 FB 134
BEGIN
   S703_TL_DC_PIN.Enable_Aux := FALSE;
   S703_TL_DC_PIN.Adv_Amount := 0;
   S703_TL_DC_PIN.Ret_Amount := 0;
   S703_TL_DC_PIN.LS_Adv1 := FALSE;
   S703_TL_DC_PIN.LS_Ret1 := FALSE;
   S703_TL_DC_PIN.LS_Adv2 := FALSE;
   S703_TL_DC_PIN.LS_Ret2 := FALSE;
   S703_TL_DC_PIN.LS_Adv3 := FALSE;
   S703_TL_DC_PIN.LS_Ret3 := FALSE;
   S703_TL_DC_PIN.LS_Adv4 := FALSE;
   S703_TL_DC_PIN.LS_Ret4 := FALSE;
   S703_TL_DC_PIN.LS_Adv5 := FALSE;
   S703_TL_DC_PIN.LS_Ret5 := FALSE;
   S703_TL_DC_PIN.LS_Adv6 := FALSE;
   S703_TL_DC_PIN.LS_Ret6 := FALSE;
   S703_TL_DC_PIN.LS_Adv7 := FALSE;
   S703_TL_DC_PIN.LS_Ret7 := FALSE;
   S703_TL_DC_PIN.LS_Adv8 := FALSE;
   S703_TL_DC_PIN.LS_Ret8 := FALSE;
   S703_TL_DC_PIN.SOL_Adv := FALSE;
   S703_TL_DC_PIN.SOL_Ret := FALSE;
   S703_TL_DC_PIN.M_Ready := FALSE;
   S703_TL_DC_PIN.T_CHK1 := T#0MS;
   S703_TL_DC_PIN.T_CHK2 := T#0MS;
   S703_TL_DC_PIN.PB_Lamp_CHK := FALSE;
   S703_TL_DC_PIN.PB_Error_Rst := FALSE;
   S703_TL_DC_PIN.M_FLICK := FALSE;
   S703_TL_DC_PIN.M_Adv_Err := FALSE;
   S703_TL_DC_PIN.M_Ret_Err := FALSE;
   S703_TL_DC_PIN.LP_Adv := FALSE;
   S703_TL_DC_PIN.LP_Ret := FALSE;
   S703_TL_DC_PIN.Visu_Adv := W#16#0;
   S703_TL_DC_PIN.Visu_Ret := W#16#0;
   S703_TL_DC_PIN.Error_T1.IN := FALSE;
   S703_TL_DC_PIN.Error_T1.PT := T#0MS;
   S703_TL_DC_PIN.Error_T1.Q := FALSE;
   S703_TL_DC_PIN.Error_T1.ET := T#0MS;
   S703_TL_DC_PIN.Error_T1.STATE := B#16#0;
   S703_TL_DC_PIN.Error_T1.STIME := T#0MS;
   S703_TL_DC_PIN.Error_T1.ATIME := T#0MS;
   S703_TL_DC_PIN.Error_T2.IN := FALSE;
   S703_TL_DC_PIN.Error_T2.PT := T#0MS;
   S703_TL_DC_PIN.Error_T2.Q := FALSE;
   S703_TL_DC_PIN.Error_T2.ET := T#0MS;
   S703_TL_DC_PIN.Error_T2.STATE := B#16#0;
   S703_TL_DC_PIN.Error_T2.STIME := T#0MS;
   S703_TL_DC_PIN.Error_T2.ATIME := T#0MS;
   S703_TL_DC_PIN.Adv_End_Aux := FALSE;
   S703_TL_DC_PIN.Ret_End_Aux := FALSE;
   S703_TL_DC_PIN.CHK_Aux1 := FALSE;
   S703_TL_DC_PIN.CHK_Aux2 := FALSE;
   S703_TL_DC_PIN.Error_T1_DN := FALSE;
   S703_TL_DC_PIN.Error_T2_DN := FALSE;
   S703_TL_DC_PIN.Adv_Memo := FALSE;
   S703_TL_DC_PIN.Visu_Adv_Arr[0] := FALSE;
   S703_TL_DC_PIN.Visu_Adv_Arr[1] := FALSE;
   S703_TL_DC_PIN.Visu_Adv_Arr[2] := FALSE;
   S703_TL_DC_PIN.Visu_Adv_Arr[3] := FALSE;
   S703_TL_DC_PIN.Visu_Adv_Arr[4] := FALSE;
   S703_TL_DC_PIN.Visu_Adv_Arr[5] := FALSE;
   S703_TL_DC_PIN.Visu_Adv_Arr[6] := FALSE;
   S703_TL_DC_PIN.Visu_Adv_Arr[7] := FALSE;
   S703_TL_DC_PIN.Visu_Adv_Arr[8] := FALSE;
   S703_TL_DC_PIN.Visu_Adv_Arr[9] := FALSE;
   S703_TL_DC_PIN.Visu_Adv_Arr[10] := FALSE;
   S703_TL_DC_PIN.Visu_Adv_Arr[11] := FALSE;
   S703_TL_DC_PIN.Visu_Adv_Arr[12] := FALSE;
   S703_TL_DC_PIN.Visu_Adv_Arr[13] := FALSE;
   S703_TL_DC_PIN.Visu_Adv_Arr[14] := FALSE;
   S703_TL_DC_PIN.Visu_Adv_Arr[15] := FALSE;
   S703_TL_DC_PIN.Visu_Ret_Arr[0] := FALSE;
   S703_TL_DC_PIN.Visu_Ret_Arr[1] := FALSE;
   S703_TL_DC_PIN.Visu_Ret_Arr[2] := FALSE;
   S703_TL_DC_PIN.Visu_Ret_Arr[3] := FALSE;
   S703_TL_DC_PIN.Visu_Ret_Arr[4] := FALSE;
   S703_TL_DC_PIN.Visu_Ret_Arr[5] := FALSE;
   S703_TL_DC_PIN.Visu_Ret_Arr[6] := FALSE;
   S703_TL_DC_PIN.Visu_Ret_Arr[7] := FALSE;
   S703_TL_DC_PIN.Visu_Ret_Arr[8] := FALSE;
   S703_TL_DC_PIN.Visu_Ret_Arr[9] := FALSE;
   S703_TL_DC_PIN.Visu_Ret_Arr[10] := FALSE;
   S703_TL_DC_PIN.Visu_Ret_Arr[11] := FALSE;
   S703_TL_DC_PIN.Visu_Ret_Arr[12] := FALSE;
   S703_TL_DC_PIN.Visu_Ret_Arr[13] := FALSE;
   S703_TL_DC_PIN.Visu_Ret_Arr[14] := FALSE;
   S703_TL_DC_PIN.Visu_Ret_Arr[15] := FALSE;
   S703_TL_DC_PIN.BLK_Move_Ret := 0;
   S703_TL_DC_PIN.Enable := FALSE;
   S703_TL_DC_PIN.Adv_End := FALSE;
   S703_TL_DC_PIN.Ret_End := FALSE;
   S703_TL_DC_LATCH1.Enable_Aux := FALSE;
   S703_TL_DC_LATCH1.Adv_Amount := 0;
   S703_TL_DC_LATCH1.Ret_Amount := 0;
   S703_TL_DC_LATCH1.LS_Adv1 := FALSE;
   S703_TL_DC_LATCH1.LS_Ret1 := FALSE;
   S703_TL_DC_LATCH1.LS_Adv2 := FALSE;
   S703_TL_DC_LATCH1.LS_Ret2 := FALSE;
   S703_TL_DC_LATCH1.LS_Adv3 := FALSE;
   S703_TL_DC_LATCH1.LS_Ret3 := FALSE;
   S703_TL_DC_LATCH1.LS_Adv4 := FALSE;
   S703_TL_DC_LATCH1.LS_Ret4 := FALSE;
   S703_TL_DC_LATCH1.LS_Adv5 := FALSE;
   S703_TL_DC_LATCH1.LS_Ret5 := FALSE;
   S703_TL_DC_LATCH1.LS_Adv6 := FALSE;
   S703_TL_DC_LATCH1.LS_Ret6 := FALSE;
   S703_TL_DC_LATCH1.LS_Adv7 := FALSE;
   S703_TL_DC_LATCH1.LS_Ret7 := FALSE;
   S703_TL_DC_LATCH1.LS_Adv8 := FALSE;
   S703_TL_DC_LATCH1.LS_Ret8 := FALSE;
   S703_TL_DC_LATCH1.SOL_Adv := FALSE;
   S703_TL_DC_LATCH1.SOL_Ret := FALSE;
   S703_TL_DC_LATCH1.M_Ready := FALSE;
   S703_TL_DC_LATCH1.T_CHK1 := T#0MS;
   S703_TL_DC_LATCH1.T_CHK2 := T#0MS;
   S703_TL_DC_LATCH1.PB_Lamp_CHK := FALSE;
   S703_TL_DC_LATCH1.PB_Error_Rst := FALSE;
   S703_TL_DC_LATCH1.M_FLICK := FALSE;
   S703_TL_DC_LATCH1.M_Adv_Err := FALSE;
   S703_TL_DC_LATCH1.M_Ret_Err := FALSE;
   S703_TL_DC_LATCH1.LP_Adv := FALSE;
   S703_TL_DC_LATCH1.LP_Ret := FALSE;
   S703_TL_DC_LATCH1.Visu_Adv := W#16#0;
   S703_TL_DC_LATCH1.Visu_Ret := W#16#0;
   S703_TL_DC_LATCH1.Error_T1.IN := FALSE;
   S703_TL_DC_LATCH1.Error_T1.PT := T#0MS;
   S703_TL_DC_LATCH1.Error_T1.Q := FALSE;
   S703_TL_DC_LATCH1.Error_T1.ET := T#0MS;
   S703_TL_DC_LATCH1.Error_T1.STATE := B#16#0;
   S703_TL_DC_LATCH1.Error_T1.STIME := T#0MS;
   S703_TL_DC_LATCH1.Error_T1.ATIME := T#0MS;
   S703_TL_DC_LATCH1.Error_T2.IN := FALSE;
   S703_TL_DC_LATCH1.Error_T2.PT := T#0MS;
   S703_TL_DC_LATCH1.Error_T2.Q := FALSE;
   S703_TL_DC_LATCH1.Error_T2.ET := T#0MS;
   S703_TL_DC_LATCH1.Error_T2.STATE := B#16#0;
   S703_TL_DC_LATCH1.Error_T2.STIME := T#0MS;
   S703_TL_DC_LATCH1.Error_T2.ATIME := T#0MS;
   S703_TL_DC_LATCH1.Adv_End_Aux := FALSE;
   S703_TL_DC_LATCH1.Ret_End_Aux := FALSE;
   S703_TL_DC_LATCH1.CHK_Aux1 := FALSE;
   S703_TL_DC_LATCH1.CHK_Aux2 := FALSE;
   S703_TL_DC_LATCH1.Error_T1_DN := FALSE;
   S703_TL_DC_LATCH1.Error_T2_DN := FALSE;
   S703_TL_DC_LATCH1.Adv_Memo := FALSE;
   S703_TL_DC_LATCH1.Visu_Adv_Arr[0] := FALSE;
   S703_TL_DC_LATCH1.Visu_Adv_Arr[1] := FALSE;
   S703_TL_DC_LATCH1.Visu_Adv_Arr[2] := FALSE;
   S703_TL_DC_LATCH1.Visu_Adv_Arr[3] := FALSE;
   S703_TL_DC_LATCH1.Visu_Adv_Arr[4] := FALSE;
   S703_TL_DC_LATCH1.Visu_Adv_Arr[5] := FALSE;
   S703_TL_DC_LATCH1.Visu_Adv_Arr[6] := FALSE;
   S703_TL_DC_LATCH1.Visu_Adv_Arr[7] := FALSE;
   S703_TL_DC_LATCH1.Visu_Adv_Arr[8] := FALSE;
   S703_TL_DC_LATCH1.Visu_Adv_Arr[9] := FALSE;
   S703_TL_DC_LATCH1.Visu_Adv_Arr[10] := FALSE;
   S703_TL_DC_LATCH1.Visu_Adv_Arr[11] := FALSE;
   S703_TL_DC_LATCH1.Visu_Adv_Arr[12] := FALSE;
   S703_TL_DC_LATCH1.Visu_Adv_Arr[13] := FALSE;
   S703_TL_DC_LATCH1.Visu_Adv_Arr[14] := FALSE;
   S703_TL_DC_LATCH1.Visu_Adv_Arr[15] := FALSE;
   S703_TL_DC_LATCH1.Visu_Ret_Arr[0] := FALSE;
   S703_TL_DC_LATCH1.Visu_Ret_Arr[1] := FALSE;
   S703_TL_DC_LATCH1.Visu_Ret_Arr[2] := FALSE;
   S703_TL_DC_LATCH1.Visu_Ret_Arr[3] := FALSE;
   S703_TL_DC_LATCH1.Visu_Ret_Arr[4] := FALSE;
   S703_TL_DC_LATCH1.Visu_Ret_Arr[5] := FALSE;
   S703_TL_DC_LATCH1.Visu_Ret_Arr[6] := FALSE;
   S703_TL_DC_LATCH1.Visu_Ret_Arr[7] := FALSE;
   S703_TL_DC_LATCH1.Visu_Ret_Arr[8] := FALSE;
   S703_TL_DC_LATCH1.Visu_Ret_Arr[9] := FALSE;
   S703_TL_DC_LATCH1.Visu_Ret_Arr[10] := FALSE;
   S703_TL_DC_LATCH1.Visu_Ret_Arr[11] := FALSE;
   S703_TL_DC_LATCH1.Visu_Ret_Arr[12] := FALSE;
   S703_TL_DC_LATCH1.Visu_Ret_Arr[13] := FALSE;
   S703_TL_DC_LATCH1.Visu_Ret_Arr[14] := FALSE;
   S703_TL_DC_LATCH1.Visu_Ret_Arr[15] := FALSE;
   S703_TL_DC_LATCH1.BLK_Move_Ret := 0;
   S703_TL_DC_LATCH1.Enable := FALSE;
   S703_TL_DC_LATCH1.Adv_End := FALSE;
   S703_TL_DC_LATCH1.Ret_End := FALSE;
   S703_TL_DC_LATCH2.Enable_Aux := FALSE;
   S703_TL_DC_LATCH2.Adv_Amount := 0;
   S703_TL_DC_LATCH2.Ret_Amount := 0;
   S703_TL_DC_LATCH2.LS_Adv1 := FALSE;
   S703_TL_DC_LATCH2.LS_Ret1 := FALSE;
   S703_TL_DC_LATCH2.LS_Adv2 := FALSE;
   S703_TL_DC_LATCH2.LS_Ret2 := FALSE;
   S703_TL_DC_LATCH2.LS_Adv3 := FALSE;
   S703_TL_DC_LATCH2.LS_Ret3 := FALSE;
   S703_TL_DC_LATCH2.LS_Adv4 := FALSE;
   S703_TL_DC_LATCH2.LS_Ret4 := FALSE;
   S703_TL_DC_LATCH2.LS_Adv5 := FALSE;
   S703_TL_DC_LATCH2.LS_Ret5 := FALSE;
   S703_TL_DC_LATCH2.LS_Adv6 := FALSE;
   S703_TL_DC_LATCH2.LS_Ret6 := FALSE;
   S703_TL_DC_LATCH2.LS_Adv7 := FALSE;
   S703_TL_DC_LATCH2.LS_Ret7 := FALSE;
   S703_TL_DC_LATCH2.LS_Adv8 := FALSE;
   S703_TL_DC_LATCH2.LS_Ret8 := FALSE;
   S703_TL_DC_LATCH2.SOL_Adv := FALSE;
   S703_TL_DC_LATCH2.SOL_Ret := FALSE;
   S703_TL_DC_LATCH2.M_Ready := FALSE;
   S703_TL_DC_LATCH2.T_CHK1 := T#0MS;
   S703_TL_DC_LATCH2.T_CHK2 := T#0MS;
   S703_TL_DC_LATCH2.PB_Lamp_CHK := FALSE;
   S703_TL_DC_LATCH2.PB_Error_Rst := FALSE;
   S703_TL_DC_LATCH2.M_FLICK := FALSE;
   S703_TL_DC_LATCH2.M_Adv_Err := FALSE;
   S703_TL_DC_LATCH2.M_Ret_Err := FALSE;
   S703_TL_DC_LATCH2.LP_Adv := FALSE;
   S703_TL_DC_LATCH2.LP_Ret := FALSE;
   S703_TL_DC_LATCH2.Visu_Adv := W#16#0;
   S703_TL_DC_LATCH2.Visu_Ret := W#16#0;
   S703_TL_DC_LATCH2.Error_T1.IN := FALSE;
   S703_TL_DC_LATCH2.Error_T1.PT := T#0MS;
   S703_TL_DC_LATCH2.Error_T1.Q := FALSE;
   S703_TL_DC_LATCH2.Error_T1.ET := T#0MS;
   S703_TL_DC_LATCH2.Error_T1.STATE := B#16#0;
   S703_TL_DC_LATCH2.Error_T1.STIME := T#0MS;
   S703_TL_DC_LATCH2.Error_T1.ATIME := T#0MS;
   S703_TL_DC_LATCH2.Error_T2.IN := FALSE;
   S703_TL_DC_LATCH2.Error_T2.PT := T#0MS;
   S703_TL_DC_LATCH2.Error_T2.Q := FALSE;
   S703_TL_DC_LATCH2.Error_T2.ET := T#0MS;
   S703_TL_DC_LATCH2.Error_T2.STATE := B#16#0;
   S703_TL_DC_LATCH2.Error_T2.STIME := T#0MS;
   S703_TL_DC_LATCH2.Error_T2.ATIME := T#0MS;
   S703_TL_DC_LATCH2.Adv_End_Aux := FALSE;
   S703_TL_DC_LATCH2.Ret_End_Aux := FALSE;
   S703_TL_DC_LATCH2.CHK_Aux1 := FALSE;
   S703_TL_DC_LATCH2.CHK_Aux2 := FALSE;
   S703_TL_DC_LATCH2.Error_T1_DN := FALSE;
   S703_TL_DC_LATCH2.Error_T2_DN := FALSE;
   S703_TL_DC_LATCH2.Adv_Memo := FALSE;
   S703_TL_DC_LATCH2.Visu_Adv_Arr[0] := FALSE;
   S703_TL_DC_LATCH2.Visu_Adv_Arr[1] := FALSE;
   S703_TL_DC_LATCH2.Visu_Adv_Arr[2] := FALSE;
   S703_TL_DC_LATCH2.Visu_Adv_Arr[3] := FALSE;
   S703_TL_DC_LATCH2.Visu_Adv_Arr[4] := FALSE;
   S703_TL_DC_LATCH2.Visu_Adv_Arr[5] := FALSE;
   S703_TL_DC_LATCH2.Visu_Adv_Arr[6] := FALSE;
   S703_TL_DC_LATCH2.Visu_Adv_Arr[7] := FALSE;
   S703_TL_DC_LATCH2.Visu_Adv_Arr[8] := FALSE;
   S703_TL_DC_LATCH2.Visu_Adv_Arr[9] := FALSE;
   S703_TL_DC_LATCH2.Visu_Adv_Arr[10] := FALSE;
   S703_TL_DC_LATCH2.Visu_Adv_Arr[11] := FALSE;
   S703_TL_DC_LATCH2.Visu_Adv_Arr[12] := FALSE;
   S703_TL_DC_LATCH2.Visu_Adv_Arr[13] := FALSE;
   S703_TL_DC_LATCH2.Visu_Adv_Arr[14] := FALSE;
   S703_TL_DC_LATCH2.Visu_Adv_Arr[15] := FALSE;
   S703_TL_DC_LATCH2.Visu_Ret_Arr[0] := FALSE;
   S703_TL_DC_LATCH2.Visu_Ret_Arr[1] := FALSE;
   S703_TL_DC_LATCH2.Visu_Ret_Arr[2] := FALSE;
   S703_TL_DC_LATCH2.Visu_Ret_Arr[3] := FALSE;
   S703_TL_DC_LATCH2.Visu_Ret_Arr[4] := FALSE;
   S703_TL_DC_LATCH2.Visu_Ret_Arr[5] := FALSE;
   S703_TL_DC_LATCH2.Visu_Ret_Arr[6] := FALSE;
   S703_TL_DC_LATCH2.Visu_Ret_Arr[7] := FALSE;
   S703_TL_DC_LATCH2.Visu_Ret_Arr[8] := FALSE;
   S703_TL_DC_LATCH2.Visu_Ret_Arr[9] := FALSE;
   S703_TL_DC_LATCH2.Visu_Ret_Arr[10] := FALSE;
   S703_TL_DC_LATCH2.Visu_Ret_Arr[11] := FALSE;
   S703_TL_DC_LATCH2.Visu_Ret_Arr[12] := FALSE;
   S703_TL_DC_LATCH2.Visu_Ret_Arr[13] := FALSE;
   S703_TL_DC_LATCH2.Visu_Ret_Arr[14] := FALSE;
   S703_TL_DC_LATCH2.Visu_Ret_Arr[15] := FALSE;
   S703_TL_DC_LATCH2.BLK_Move_Ret := 0;
   S703_TL_DC_LATCH2.Enable := FALSE;
   S703_TL_DC_LATCH2.Adv_End := FALSE;
   S703_TL_DC_LATCH2.Ret_End := FALSE;
   S703_TL_DC_1ST_CLAMP1.Enable_Aux := FALSE;
   S703_TL_DC_1ST_CLAMP1.Adv_Amount := 0;
   S703_TL_DC_1ST_CLAMP1.Ret_Amount := 0;
   S703_TL_DC_1ST_CLAMP1.LS_Adv1 := FALSE;
   S703_TL_DC_1ST_CLAMP1.LS_Ret1 := FALSE;
   S703_TL_DC_1ST_CLAMP1.LS_Adv2 := FALSE;
   S703_TL_DC_1ST_CLAMP1.LS_Ret2 := FALSE;
   S703_TL_DC_1ST_CLAMP1.LS_Adv3 := FALSE;
   S703_TL_DC_1ST_CLAMP1.LS_Ret3 := FALSE;
   S703_TL_DC_1ST_CLAMP1.LS_Adv4 := FALSE;
   S703_TL_DC_1ST_CLAMP1.LS_Ret4 := FALSE;
   S703_TL_DC_1ST_CLAMP1.LS_Adv5 := FALSE;
   S703_TL_DC_1ST_CLAMP1.LS_Ret5 := FALSE;
   S703_TL_DC_1ST_CLAMP1.LS_Adv6 := FALSE;
   S703_TL_DC_1ST_CLAMP1.LS_Ret6 := FALSE;
   S703_TL_DC_1ST_CLAMP1.LS_Adv7 := FALSE;
   S703_TL_DC_1ST_CLAMP1.LS_Ret7 := FALSE;
   S703_TL_DC_1ST_CLAMP1.LS_Adv8 := FALSE;
   S703_TL_DC_1ST_CLAMP1.LS_Ret8 := FALSE;
   S703_TL_DC_1ST_CLAMP1.SOL_Adv := FALSE;
   S703_TL_DC_1ST_CLAMP1.SOL_Ret := FALSE;
   S703_TL_DC_1ST_CLAMP1.M_Ready := FALSE;
   S703_TL_DC_1ST_CLAMP1.T_CHK1 := T#0MS;
   S703_TL_DC_1ST_CLAMP1.T_CHK2 := T#0MS;
   S703_TL_DC_1ST_CLAMP1.PB_Lamp_CHK := FALSE;
   S703_TL_DC_1ST_CLAMP1.PB_Error_Rst := FALSE;
   S703_TL_DC_1ST_CLAMP1.M_FLICK := FALSE;
   S703_TL_DC_1ST_CLAMP1.M_Adv_Err := FALSE;
   S703_TL_DC_1ST_CLAMP1.M_Ret_Err := FALSE;
   S703_TL_DC_1ST_CLAMP1.LP_Adv := FALSE;
   S703_TL_DC_1ST_CLAMP1.LP_Ret := FALSE;
   S703_TL_DC_1ST_CLAMP1.Visu_Adv := W#16#0;
   S703_TL_DC_1ST_CLAMP1.Visu_Ret := W#16#0;
   S703_TL_DC_1ST_CLAMP1.Error_T1.IN := FALSE;
   S703_TL_DC_1ST_CLAMP1.Error_T1.PT := T#0MS;
   S703_TL_DC_1ST_CLAMP1.Error_T1.Q := FALSE;
   S703_TL_DC_1ST_CLAMP1.Error_T1.ET := T#0MS;
   S703_TL_DC_1ST_CLAMP1.Error_T1.STATE := B#16#0;
   S703_TL_DC_1ST_CLAMP1.Error_T1.STIME := T#0MS;
   S703_TL_DC_1ST_CLAMP1.Error_T1.ATIME := T#0MS;
   S703_TL_DC_1ST_CLAMP1.Error_T2.IN := FALSE;
   S703_TL_DC_1ST_CLAMP1.Error_T2.PT := T#0MS;
   S703_TL_DC_1ST_CLAMP1.Error_T2.Q := FALSE;
   S703_TL_DC_1ST_CLAMP1.Error_T2.ET := T#0MS;
   S703_TL_DC_1ST_CLAMP1.Error_T2.STATE := B#16#0;
   S703_TL_DC_1ST_CLAMP1.Error_T2.STIME := T#0MS;
   S703_TL_DC_1ST_CLAMP1.Error_T2.ATIME := T#0MS;
   S703_TL_DC_1ST_CLAMP1.Adv_End_Aux := FALSE;
   S703_TL_DC_1ST_CLAMP1.Ret_End_Aux := FALSE;
   S703_TL_DC_1ST_CLAMP1.CHK_Aux1 := FALSE;
   S703_TL_DC_1ST_CLAMP1.CHK_Aux2 := FALSE;
   S703_TL_DC_1ST_CLAMP1.Error_T1_DN := FALSE;
   S703_TL_DC_1ST_CLAMP1.Error_T2_DN := FALSE;
   S703_TL_DC_1ST_CLAMP1.Adv_Memo := FALSE;
   S703_TL_DC_1ST_CLAMP1.Visu_Adv_Arr[0] := FALSE;
   S703_TL_DC_1ST_CLAMP1.Visu_Adv_Arr[1] := FALSE;
   S703_TL_DC_1ST_CLAMP1.Visu_Adv_Arr[2] := FALSE;
   S703_TL_DC_1ST_CLAMP1.Visu_Adv_Arr[3] := FALSE;
   S703_TL_DC_1ST_CLAMP1.Visu_Adv_Arr[4] := FALSE;
   S703_TL_DC_1ST_CLAMP1.Visu_Adv_Arr[5] := FALSE;
   S703_TL_DC_1ST_CLAMP1.Visu_Adv_Arr[6] := FALSE;
   S703_TL_DC_1ST_CLAMP1.Visu_Adv_Arr[7] := FALSE;
   S703_TL_DC_1ST_CLAMP1.Visu_Adv_Arr[8] := FALSE;
   S703_TL_DC_1ST_CLAMP1.Visu_Adv_Arr[9] := FALSE;
   S703_TL_DC_1ST_CLAMP1.Visu_Adv_Arr[10] := FALSE;
   S703_TL_DC_1ST_CLAMP1.Visu_Adv_Arr[11] := FALSE;
   S703_TL_DC_1ST_CLAMP1.Visu_Adv_Arr[12] := FALSE;
   S703_TL_DC_1ST_CLAMP1.Visu_Adv_Arr[13] := FALSE;
   S703_TL_DC_1ST_CLAMP1.Visu_Adv_Arr[14] := FALSE;
   S703_TL_DC_1ST_CLAMP1.Visu_Adv_Arr[15] := FALSE;
   S703_TL_DC_1ST_CLAMP1.Visu_Ret_Arr[0] := FALSE;
   S703_TL_DC_1ST_CLAMP1.Visu_Ret_Arr[1] := FALSE;
   S703_TL_DC_1ST_CLAMP1.Visu_Ret_Arr[2] := FALSE;
   S703_TL_DC_1ST_CLAMP1.Visu_Ret_Arr[3] := FALSE;
   S703_TL_DC_1ST_CLAMP1.Visu_Ret_Arr[4] := FALSE;
   S703_TL_DC_1ST_CLAMP1.Visu_Ret_Arr[5] := FALSE;
   S703_TL_DC_1ST_CLAMP1.Visu_Ret_Arr[6] := FALSE;
   S703_TL_DC_1ST_CLAMP1.Visu_Ret_Arr[7] := FALSE;
   S703_TL_DC_1ST_CLAMP1.Visu_Ret_Arr[8] := FALSE;
   S703_TL_DC_1ST_CLAMP1.Visu_Ret_Arr[9] := FALSE;
   S703_TL_DC_1ST_CLAMP1.Visu_Ret_Arr[10] := FALSE;
   S703_TL_DC_1ST_CLAMP1.Visu_Ret_Arr[11] := FALSE;
   S703_TL_DC_1ST_CLAMP1.Visu_Ret_Arr[12] := FALSE;
   S703_TL_DC_1ST_CLAMP1.Visu_Ret_Arr[13] := FALSE;
   S703_TL_DC_1ST_CLAMP1.Visu_Ret_Arr[14] := FALSE;
   S703_TL_DC_1ST_CLAMP1.Visu_Ret_Arr[15] := FALSE;
   S703_TL_DC_1ST_CLAMP1.BLK_Move_Ret := 0;
   S703_TL_DC_1ST_CLAMP1.Enable := FALSE;
   S703_TL_DC_1ST_CLAMP1.Adv_End := FALSE;
   S703_TL_DC_1ST_CLAMP1.Ret_End := FALSE;
   S703_TL_DC_1ST_CLAMP2.Enable_Aux := FALSE;
   S703_TL_DC_1ST_CLAMP2.Adv_Amount := 0;
   S703_TL_DC_1ST_CLAMP2.Ret_Amount := 0;
   S703_TL_DC_1ST_CLAMP2.LS_Adv1 := FALSE;
   S703_TL_DC_1ST_CLAMP2.LS_Ret1 := FALSE;
   S703_TL_DC_1ST_CLAMP2.LS_Adv2 := FALSE;
   S703_TL_DC_1ST_CLAMP2.LS_Ret2 := FALSE;
   S703_TL_DC_1ST_CLAMP2.LS_Adv3 := FALSE;
   S703_TL_DC_1ST_CLAMP2.LS_Ret3 := FALSE;
   S703_TL_DC_1ST_CLAMP2.LS_Adv4 := FALSE;
   S703_TL_DC_1ST_CLAMP2.LS_Ret4 := FALSE;
   S703_TL_DC_1ST_CLAMP2.LS_Adv5 := FALSE;
   S703_TL_DC_1ST_CLAMP2.LS_Ret5 := FALSE;
   S703_TL_DC_1ST_CLAMP2.LS_Adv6 := FALSE;
   S703_TL_DC_1ST_CLAMP2.LS_Ret6 := FALSE;
   S703_TL_DC_1ST_CLAMP2.LS_Adv7 := FALSE;
   S703_TL_DC_1ST_CLAMP2.LS_Ret7 := FALSE;
   S703_TL_DC_1ST_CLAMP2.LS_Adv8 := FALSE;
   S703_TL_DC_1ST_CLAMP2.LS_Ret8 := FALSE;
   S703_TL_DC_1ST_CLAMP2.SOL_Adv := FALSE;
   S703_TL_DC_1ST_CLAMP2.SOL_Ret := FALSE;
   S703_TL_DC_1ST_CLAMP2.M_Ready := FALSE;
   S703_TL_DC_1ST_CLAMP2.T_CHK1 := T#0MS;
   S703_TL_DC_1ST_CLAMP2.T_CHK2 := T#0MS;
   S703_TL_DC_1ST_CLAMP2.PB_Lamp_CHK := FALSE;
   S703_TL_DC_1ST_CLAMP2.PB_Error_Rst := FALSE;
   S703_TL_DC_1ST_CLAMP2.M_FLICK := FALSE;
   S703_TL_DC_1ST_CLAMP2.M_Adv_Err := FALSE;
   S703_TL_DC_1ST_CLAMP2.M_Ret_Err := FALSE;
   S703_TL_DC_1ST_CLAMP2.LP_Adv := FALSE;
   S703_TL_DC_1ST_CLAMP2.LP_Ret := FALSE;
   S703_TL_DC_1ST_CLAMP2.Visu_Adv := W#16#0;
   S703_TL_DC_1ST_CLAMP2.Visu_Ret := W#16#0;
   S703_TL_DC_1ST_CLAMP2.Error_T1.IN := FALSE;
   S703_TL_DC_1ST_CLAMP2.Error_T1.PT := T#0MS;
   S703_TL_DC_1ST_CLAMP2.Error_T1.Q := FALSE;
   S703_TL_DC_1ST_CLAMP2.Error_T1.ET := T#0MS;
   S703_TL_DC_1ST_CLAMP2.Error_T1.STATE := B#16#0;
   S703_TL_DC_1ST_CLAMP2.Error_T1.STIME := T#0MS;
   S703_TL_DC_1ST_CLAMP2.Error_T1.ATIME := T#0MS;
   S703_TL_DC_1ST_CLAMP2.Error_T2.IN := FALSE;
   S703_TL_DC_1ST_CLAMP2.Error_T2.PT := T#0MS;
   S703_TL_DC_1ST_CLAMP2.Error_T2.Q := FALSE;
   S703_TL_DC_1ST_CLAMP2.Error_T2.ET := T#0MS;
   S703_TL_DC_1ST_CLAMP2.Error_T2.STATE := B#16#0;
   S703_TL_DC_1ST_CLAMP2.Error_T2.STIME := T#0MS;
   S703_TL_DC_1ST_CLAMP2.Error_T2.ATIME := T#0MS;
   S703_TL_DC_1ST_CLAMP2.Adv_End_Aux := FALSE;
   S703_TL_DC_1ST_CLAMP2.Ret_End_Aux := FALSE;
   S703_TL_DC_1ST_CLAMP2.CHK_Aux1 := FALSE;
   S703_TL_DC_1ST_CLAMP2.CHK_Aux2 := FALSE;
   S703_TL_DC_1ST_CLAMP2.Error_T1_DN := FALSE;
   S703_TL_DC_1ST_CLAMP2.Error_T2_DN := FALSE;
   S703_TL_DC_1ST_CLAMP2.Adv_Memo := FALSE;
   S703_TL_DC_1ST_CLAMP2.Visu_Adv_Arr[0] := FALSE;
   S703_TL_DC_1ST_CLAMP2.Visu_Adv_Arr[1] := FALSE;
   S703_TL_DC_1ST_CLAMP2.Visu_Adv_Arr[2] := FALSE;
   S703_TL_DC_1ST_CLAMP2.Visu_Adv_Arr[3] := FALSE;
   S703_TL_DC_1ST_CLAMP2.Visu_Adv_Arr[4] := FALSE;
   S703_TL_DC_1ST_CLAMP2.Visu_Adv_Arr[5] := FALSE;
   S703_TL_DC_1ST_CLAMP2.Visu_Adv_Arr[6] := FALSE;
   S703_TL_DC_1ST_CLAMP2.Visu_Adv_Arr[7] := FALSE;
   S703_TL_DC_1ST_CLAMP2.Visu_Adv_Arr[8] := FALSE;
   S703_TL_DC_1ST_CLAMP2.Visu_Adv_Arr[9] := FALSE;
   S703_TL_DC_1ST_CLAMP2.Visu_Adv_Arr[10] := FALSE;
   S703_TL_DC_1ST_CLAMP2.Visu_Adv_Arr[11] := FALSE;
   S703_TL_DC_1ST_CLAMP2.Visu_Adv_Arr[12] := FALSE;
   S703_TL_DC_1ST_CLAMP2.Visu_Adv_Arr[13] := FALSE;
   S703_TL_DC_1ST_CLAMP2.Visu_Adv_Arr[14] := FALSE;
   S703_TL_DC_1ST_CLAMP2.Visu_Adv_Arr[15] := FALSE;
   S703_TL_DC_1ST_CLAMP2.Visu_Ret_Arr[0] := FALSE;
   S703_TL_DC_1ST_CLAMP2.Visu_Ret_Arr[1] := FALSE;
   S703_TL_DC_1ST_CLAMP2.Visu_Ret_Arr[2] := FALSE;
   S703_TL_DC_1ST_CLAMP2.Visu_Ret_Arr[3] := FALSE;
   S703_TL_DC_1ST_CLAMP2.Visu_Ret_Arr[4] := FALSE;
   S703_TL_DC_1ST_CLAMP2.Visu_Ret_Arr[5] := FALSE;
   S703_TL_DC_1ST_CLAMP2.Visu_Ret_Arr[6] := FALSE;
   S703_TL_DC_1ST_CLAMP2.Visu_Ret_Arr[7] := FALSE;
   S703_TL_DC_1ST_CLAMP2.Visu_Ret_Arr[8] := FALSE;
   S703_TL_DC_1ST_CLAMP2.Visu_Ret_Arr[9] := FALSE;
   S703_TL_DC_1ST_CLAMP2.Visu_Ret_Arr[10] := FALSE;
   S703_TL_DC_1ST_CLAMP2.Visu_Ret_Arr[11] := FALSE;
   S703_TL_DC_1ST_CLAMP2.Visu_Ret_Arr[12] := FALSE;
   S703_TL_DC_1ST_CLAMP2.Visu_Ret_Arr[13] := FALSE;
   S703_TL_DC_1ST_CLAMP2.Visu_Ret_Arr[14] := FALSE;
   S703_TL_DC_1ST_CLAMP2.Visu_Ret_Arr[15] := FALSE;
   S703_TL_DC_1ST_CLAMP2.BLK_Move_Ret := 0;
   S703_TL_DC_1ST_CLAMP2.Enable := FALSE;
   S703_TL_DC_1ST_CLAMP2.Adv_End := FALSE;
   S703_TL_DC_1ST_CLAMP2.Ret_End := FALSE;
   S703_TL_DC_1ST_CLAMP3.Enable_Aux := FALSE;
   S703_TL_DC_1ST_CLAMP3.Adv_Amount := 0;
   S703_TL_DC_1ST_CLAMP3.Ret_Amount := 0;
   S703_TL_DC_1ST_CLAMP3.LS_Adv1 := FALSE;
   S703_TL_DC_1ST_CLAMP3.LS_Ret1 := FALSE;
   S703_TL_DC_1ST_CLAMP3.LS_Adv2 := FALSE;
   S703_TL_DC_1ST_CLAMP3.LS_Ret2 := FALSE;
   S703_TL_DC_1ST_CLAMP3.LS_Adv3 := FALSE;
   S703_TL_DC_1ST_CLAMP3.LS_Ret3 := FALSE;
   S703_TL_DC_1ST_CLAMP3.LS_Adv4 := FALSE;
   S703_TL_DC_1ST_CLAMP3.LS_Ret4 := FALSE;
   S703_TL_DC_1ST_CLAMP3.LS_Adv5 := FALSE;
   S703_TL_DC_1ST_CLAMP3.LS_Ret5 := FALSE;
   S703_TL_DC_1ST_CLAMP3.LS_Adv6 := FALSE;
   S703_TL_DC_1ST_CLAMP3.LS_Ret6 := FALSE;
   S703_TL_DC_1ST_CLAMP3.LS_Adv7 := FALSE;
   S703_TL_DC_1ST_CLAMP3.LS_Ret7 := FALSE;
   S703_TL_DC_1ST_CLAMP3.LS_Adv8 := FALSE;
   S703_TL_DC_1ST_CLAMP3.LS_Ret8 := FALSE;
   S703_TL_DC_1ST_CLAMP3.SOL_Adv := FALSE;
   S703_TL_DC_1ST_CLAMP3.SOL_Ret := FALSE;
   S703_TL_DC_1ST_CLAMP3.M_Ready := FALSE;
   S703_TL_DC_1ST_CLAMP3.T_CHK1 := T#0MS;
   S703_TL_DC_1ST_CLAMP3.T_CHK2 := T#0MS;
   S703_TL_DC_1ST_CLAMP3.PB_Lamp_CHK := FALSE;
   S703_TL_DC_1ST_CLAMP3.PB_Error_Rst := FALSE;
   S703_TL_DC_1ST_CLAMP3.M_FLICK := FALSE;
   S703_TL_DC_1ST_CLAMP3.M_Adv_Err := FALSE;
   S703_TL_DC_1ST_CLAMP3.M_Ret_Err := FALSE;
   S703_TL_DC_1ST_CLAMP3.LP_Adv := FALSE;
   S703_TL_DC_1ST_CLAMP3.LP_Ret := FALSE;
   S703_TL_DC_1ST_CLAMP3.Visu_Adv := W#16#0;
   S703_TL_DC_1ST_CLAMP3.Visu_Ret := W#16#0;
   S703_TL_DC_1ST_CLAMP3.Error_T1.IN := FALSE;
   S703_TL_DC_1ST_CLAMP3.Error_T1.PT := T#0MS;
   S703_TL_DC_1ST_CLAMP3.Error_T1.Q := FALSE;
   S703_TL_DC_1ST_CLAMP3.Error_T1.ET := T#0MS;
   S703_TL_DC_1ST_CLAMP3.Error_T1.STATE := B#16#0;
   S703_TL_DC_1ST_CLAMP3.Error_T1.STIME := T#0MS;
   S703_TL_DC_1ST_CLAMP3.Error_T1.ATIME := T#0MS;
   S703_TL_DC_1ST_CLAMP3.Error_T2.IN := FALSE;
   S703_TL_DC_1ST_CLAMP3.Error_T2.PT := T#0MS;
   S703_TL_DC_1ST_CLAMP3.Error_T2.Q := FALSE;
   S703_TL_DC_1ST_CLAMP3.Error_T2.ET := T#0MS;
   S703_TL_DC_1ST_CLAMP3.Error_T2.STATE := B#16#0;
   S703_TL_DC_1ST_CLAMP3.Error_T2.STIME := T#0MS;
   S703_TL_DC_1ST_CLAMP3.Error_T2.ATIME := T#0MS;
   S703_TL_DC_1ST_CLAMP3.Adv_End_Aux := FALSE;
   S703_TL_DC_1ST_CLAMP3.Ret_End_Aux := FALSE;
   S703_TL_DC_1ST_CLAMP3.CHK_Aux1 := FALSE;
   S703_TL_DC_1ST_CLAMP3.CHK_Aux2 := FALSE;
   S703_TL_DC_1ST_CLAMP3.Error_T1_DN := FALSE;
   S703_TL_DC_1ST_CLAMP3.Error_T2_DN := FALSE;
   S703_TL_DC_1ST_CLAMP3.Adv_Memo := FALSE;
   S703_TL_DC_1ST_CLAMP3.Visu_Adv_Arr[0] := FALSE;
   S703_TL_DC_1ST_CLAMP3.Visu_Adv_Arr[1] := FALSE;
   S703_TL_DC_1ST_CLAMP3.Visu_Adv_Arr[2] := FALSE;
   S703_TL_DC_1ST_CLAMP3.Visu_Adv_Arr[3] := FALSE;
   S703_TL_DC_1ST_CLAMP3.Visu_Adv_Arr[4] := FALSE;
   S703_TL_DC_1ST_CLAMP3.Visu_Adv_Arr[5] := FALSE;
   S703_TL_DC_1ST_CLAMP3.Visu_Adv_Arr[6] := FALSE;
   S703_TL_DC_1ST_CLAMP3.Visu_Adv_Arr[7] := FALSE;
   S703_TL_DC_1ST_CLAMP3.Visu_Adv_Arr[8] := FALSE;
   S703_TL_DC_1ST_CLAMP3.Visu_Adv_Arr[9] := FALSE;
   S703_TL_DC_1ST_CLAMP3.Visu_Adv_Arr[10] := FALSE;
   S703_TL_DC_1ST_CLAMP3.Visu_Adv_Arr[11] := FALSE;
   S703_TL_DC_1ST_CLAMP3.Visu_Adv_Arr[12] := FALSE;
   S703_TL_DC_1ST_CLAMP3.Visu_Adv_Arr[13] := FALSE;
   S703_TL_DC_1ST_CLAMP3.Visu_Adv_Arr[14] := FALSE;
   S703_TL_DC_1ST_CLAMP3.Visu_Adv_Arr[15] := FALSE;
   S703_TL_DC_1ST_CLAMP3.Visu_Ret_Arr[0] := FALSE;
   S703_TL_DC_1ST_CLAMP3.Visu_Ret_Arr[1] := FALSE;
   S703_TL_DC_1ST_CLAMP3.Visu_Ret_Arr[2] := FALSE;
   S703_TL_DC_1ST_CLAMP3.Visu_Ret_Arr[3] := FALSE;
   S703_TL_DC_1ST_CLAMP3.Visu_Ret_Arr[4] := FALSE;
   S703_TL_DC_1ST_CLAMP3.Visu_Ret_Arr[5] := FALSE;
   S703_TL_DC_1ST_CLAMP3.Visu_Ret_Arr[6] := FALSE;
   S703_TL_DC_1ST_CLAMP3.Visu_Ret_Arr[7] := FALSE;
   S703_TL_DC_1ST_CLAMP3.Visu_Ret_Arr[8] := FALSE;
   S703_TL_DC_1ST_CLAMP3.Visu_Ret_Arr[9] := FALSE;
   S703_TL_DC_1ST_CLAMP3.Visu_Ret_Arr[10] := FALSE;
   S703_TL_DC_1ST_CLAMP3.Visu_Ret_Arr[11] := FALSE;
   S703_TL_DC_1ST_CLAMP3.Visu_Ret_Arr[12] := FALSE;
   S703_TL_DC_1ST_CLAMP3.Visu_Ret_Arr[13] := FALSE;
   S703_TL_DC_1ST_CLAMP3.Visu_Ret_Arr[14] := FALSE;
   S703_TL_DC_1ST_CLAMP3.Visu_Ret_Arr[15] := FALSE;
   S703_TL_DC_1ST_CLAMP3.BLK_Move_Ret := 0;
   S703_TL_DC_1ST_CLAMP3.Enable := FALSE;
   S703_TL_DC_1ST_CLAMP3.Adv_End := FALSE;
   S703_TL_DC_1ST_CLAMP3.Ret_End := FALSE;
   S703_TL_DC_2ND_CLAMP1.Enable_Aux := FALSE;
   S703_TL_DC_2ND_CLAMP1.Adv_Amount := 0;
   S703_TL_DC_2ND_CLAMP1.Ret_Amount := 0;
   S703_TL_DC_2ND_CLAMP1.LS_Adv1 := FALSE;
   S703_TL_DC_2ND_CLAMP1.LS_Ret1 := FALSE;
   S703_TL_DC_2ND_CLAMP1.LS_Adv2 := FALSE;
   S703_TL_DC_2ND_CLAMP1.LS_Ret2 := FALSE;
   S703_TL_DC_2ND_CLAMP1.LS_Adv3 := FALSE;
   S703_TL_DC_2ND_CLAMP1.LS_Ret3 := FALSE;
   S703_TL_DC_2ND_CLAMP1.LS_Adv4 := FALSE;
   S703_TL_DC_2ND_CLAMP1.LS_Ret4 := FALSE;
   S703_TL_DC_2ND_CLAMP1.LS_Adv5 := FALSE;
   S703_TL_DC_2ND_CLAMP1.LS_Ret5 := FALSE;
   S703_TL_DC_2ND_CLAMP1.LS_Adv6 := FALSE;
   S703_TL_DC_2ND_CLAMP1.LS_Ret6 := FALSE;
   S703_TL_DC_2ND_CLAMP1.LS_Adv7 := FALSE;
   S703_TL_DC_2ND_CLAMP1.LS_Ret7 := FALSE;
   S703_TL_DC_2ND_CLAMP1.LS_Adv8 := FALSE;
   S703_TL_DC_2ND_CLAMP1.LS_Ret8 := FALSE;
   S703_TL_DC_2ND_CLAMP1.SOL_Adv := FALSE;
   S703_TL_DC_2ND_CLAMP1.SOL_Ret := FALSE;
   S703_TL_DC_2ND_CLAMP1.M_Ready := FALSE;
   S703_TL_DC_2ND_CLAMP1.T_CHK1 := T#0MS;
   S703_TL_DC_2ND_CLAMP1.T_CHK2 := T#0MS;
   S703_TL_DC_2ND_CLAMP1.PB_Lamp_CHK := FALSE;
   S703_TL_DC_2ND_CLAMP1.PB_Error_Rst := FALSE;
   S703_TL_DC_2ND_CLAMP1.M_FLICK := FALSE;
   S703_TL_DC_2ND_CLAMP1.M_Adv_Err := FALSE;
   S703_TL_DC_2ND_CLAMP1.M_Ret_Err := FALSE;
   S703_TL_DC_2ND_CLAMP1.LP_Adv := FALSE;
   S703_TL_DC_2ND_CLAMP1.LP_Ret := FALSE;
   S703_TL_DC_2ND_CLAMP1.Visu_Adv := W#16#0;
   S703_TL_DC_2ND_CLAMP1.Visu_Ret := W#16#0;
   S703_TL_DC_2ND_CLAMP1.Error_T1.IN := FALSE;
   S703_TL_DC_2ND_CLAMP1.Error_T1.PT := T#0MS;
   S703_TL_DC_2ND_CLAMP1.Error_T1.Q := FALSE;
   S703_TL_DC_2ND_CLAMP1.Error_T1.ET := T#0MS;
   S703_TL_DC_2ND_CLAMP1.Error_T1.STATE := B#16#0;
   S703_TL_DC_2ND_CLAMP1.Error_T1.STIME := T#0MS;
   S703_TL_DC_2ND_CLAMP1.Error_T1.ATIME := T#0MS;
   S703_TL_DC_2ND_CLAMP1.Error_T2.IN := FALSE;
   S703_TL_DC_2ND_CLAMP1.Error_T2.PT := T#0MS;
   S703_TL_DC_2ND_CLAMP1.Error_T2.Q := FALSE;
   S703_TL_DC_2ND_CLAMP1.Error_T2.ET := T#0MS;
   S703_TL_DC_2ND_CLAMP1.Error_T2.STATE := B#16#0;
   S703_TL_DC_2ND_CLAMP1.Error_T2.STIME := T#0MS;
   S703_TL_DC_2ND_CLAMP1.Error_T2.ATIME := T#0MS;
   S703_TL_DC_2ND_CLAMP1.Adv_End_Aux := FALSE;
   S703_TL_DC_2ND_CLAMP1.Ret_End_Aux := FALSE;
   S703_TL_DC_2ND_CLAMP1.CHK_Aux1 := FALSE;
   S703_TL_DC_2ND_CLAMP1.CHK_Aux2 := FALSE;
   S703_TL_DC_2ND_CLAMP1.Error_T1_DN := FALSE;
   S703_TL_DC_2ND_CLAMP1.Error_T2_DN := FALSE;
   S703_TL_DC_2ND_CLAMP1.Adv_Memo := FALSE;
   S703_TL_DC_2ND_CLAMP1.Visu_Adv_Arr[0] := FALSE;
   S703_TL_DC_2ND_CLAMP1.Visu_Adv_Arr[1] := FALSE;
   S703_TL_DC_2ND_CLAMP1.Visu_Adv_Arr[2] := FALSE;
   S703_TL_DC_2ND_CLAMP1.Visu_Adv_Arr[3] := FALSE;
   S703_TL_DC_2ND_CLAMP1.Visu_Adv_Arr[4] := FALSE;
   S703_TL_DC_2ND_CLAMP1.Visu_Adv_Arr[5] := FALSE;
   S703_TL_DC_2ND_CLAMP1.Visu_Adv_Arr[6] := FALSE;
   S703_TL_DC_2ND_CLAMP1.Visu_Adv_Arr[7] := FALSE;
   S703_TL_DC_2ND_CLAMP1.Visu_Adv_Arr[8] := FALSE;
   S703_TL_DC_2ND_CLAMP1.Visu_Adv_Arr[9] := FALSE;
   S703_TL_DC_2ND_CLAMP1.Visu_Adv_Arr[10] := FALSE;
   S703_TL_DC_2ND_CLAMP1.Visu_Adv_Arr[11] := FALSE;
   S703_TL_DC_2ND_CLAMP1.Visu_Adv_Arr[12] := FALSE;
   S703_TL_DC_2ND_CLAMP1.Visu_Adv_Arr[13] := FALSE;
   S703_TL_DC_2ND_CLAMP1.Visu_Adv_Arr[14] := FALSE;
   S703_TL_DC_2ND_CLAMP1.Visu_Adv_Arr[15] := FALSE;
   S703_TL_DC_2ND_CLAMP1.Visu_Ret_Arr[0] := FALSE;
   S703_TL_DC_2ND_CLAMP1.Visu_Ret_Arr[1] := FALSE;
   S703_TL_DC_2ND_CLAMP1.Visu_Ret_Arr[2] := FALSE;
   S703_TL_DC_2ND_CLAMP1.Visu_Ret_Arr[3] := FALSE;
   S703_TL_DC_2ND_CLAMP1.Visu_Ret_Arr[4] := FALSE;
   S703_TL_DC_2ND_CLAMP1.Visu_Ret_Arr[5] := FALSE;
   S703_TL_DC_2ND_CLAMP1.Visu_Ret_Arr[6] := FALSE;
   S703_TL_DC_2ND_CLAMP1.Visu_Ret_Arr[7] := FALSE;
   S703_TL_DC_2ND_CLAMP1.Visu_Ret_Arr[8] := FALSE;
   S703_TL_DC_2ND_CLAMP1.Visu_Ret_Arr[9] := FALSE;
   S703_TL_DC_2ND_CLAMP1.Visu_Ret_Arr[10] := FALSE;
   S703_TL_DC_2ND_CLAMP1.Visu_Ret_Arr[11] := FALSE;
   S703_TL_DC_2ND_CLAMP1.Visu_Ret_Arr[12] := FALSE;
   S703_TL_DC_2ND_CLAMP1.Visu_Ret_Arr[13] := FALSE;
   S703_TL_DC_2ND_CLAMP1.Visu_Ret_Arr[14] := FALSE;
   S703_TL_DC_2ND_CLAMP1.Visu_Ret_Arr[15] := FALSE;
   S703_TL_DC_2ND_CLAMP1.BLK_Move_Ret := 0;
   S703_TL_DC_2ND_CLAMP1.Enable := FALSE;
   S703_TL_DC_2ND_CLAMP1.Adv_End := FALSE;
   S703_TL_DC_2ND_CLAMP1.Ret_End := FALSE;
   S703_TL_DC_2ND_CLAMP2.Enable_Aux := FALSE;
   S703_TL_DC_2ND_CLAMP2.Adv_Amount := 0;
   S703_TL_DC_2ND_CLAMP2.Ret_Amount := 0;
   S703_TL_DC_2ND_CLAMP2.LS_Adv1 := FALSE;
   S703_TL_DC_2ND_CLAMP2.LS_Ret1 := FALSE;
   S703_TL_DC_2ND_CLAMP2.LS_Adv2 := FALSE;
   S703_TL_DC_2ND_CLAMP2.LS_Ret2 := FALSE;
   S703_TL_DC_2ND_CLAMP2.LS_Adv3 := FALSE;
   S703_TL_DC_2ND_CLAMP2.LS_Ret3 := FALSE;
   S703_TL_DC_2ND_CLAMP2.LS_Adv4 := FALSE;
   S703_TL_DC_2ND_CLAMP2.LS_Ret4 := FALSE;
   S703_TL_DC_2ND_CLAMP2.LS_Adv5 := FALSE;
   S703_TL_DC_2ND_CLAMP2.LS_Ret5 := FALSE;
   S703_TL_DC_2ND_CLAMP2.LS_Adv6 := FALSE;
   S703_TL_DC_2ND_CLAMP2.LS_Ret6 := FALSE;
   S703_TL_DC_2ND_CLAMP2.LS_Adv7 := FALSE;
   S703_TL_DC_2ND_CLAMP2.LS_Ret7 := FALSE;
   S703_TL_DC_2ND_CLAMP2.LS_Adv8 := FALSE;
   S703_TL_DC_2ND_CLAMP2.LS_Ret8 := FALSE;
   S703_TL_DC_2ND_CLAMP2.SOL_Adv := FALSE;
   S703_TL_DC_2ND_CLAMP2.SOL_Ret := FALSE;
   S703_TL_DC_2ND_CLAMP2.M_Ready := FALSE;
   S703_TL_DC_2ND_CLAMP2.T_CHK1 := T#0MS;
   S703_TL_DC_2ND_CLAMP2.T_CHK2 := T#0MS;
   S703_TL_DC_2ND_CLAMP2.PB_Lamp_CHK := FALSE;
   S703_TL_DC_2ND_CLAMP2.PB_Error_Rst := FALSE;
   S703_TL_DC_2ND_CLAMP2.M_FLICK := FALSE;
   S703_TL_DC_2ND_CLAMP2.M_Adv_Err := FALSE;
   S703_TL_DC_2ND_CLAMP2.M_Ret_Err := FALSE;
   S703_TL_DC_2ND_CLAMP2.LP_Adv := FALSE;
   S703_TL_DC_2ND_CLAMP2.LP_Ret := FALSE;
   S703_TL_DC_2ND_CLAMP2.Visu_Adv := W#16#0;
   S703_TL_DC_2ND_CLAMP2.Visu_Ret := W#16#0;
   S703_TL_DC_2ND_CLAMP2.Error_T1.IN := FALSE;
   S703_TL_DC_2ND_CLAMP2.Error_T1.PT := T#0MS;
   S703_TL_DC_2ND_CLAMP2.Error_T1.Q := FALSE;
   S703_TL_DC_2ND_CLAMP2.Error_T1.ET := T#0MS;
   S703_TL_DC_2ND_CLAMP2.Error_T1.STATE := B#16#0;
   S703_TL_DC_2ND_CLAMP2.Error_T1.STIME := T#0MS;
   S703_TL_DC_2ND_CLAMP2.Error_T1.ATIME := T#0MS;
   S703_TL_DC_2ND_CLAMP2.Error_T2.IN := FALSE;
   S703_TL_DC_2ND_CLAMP2.Error_T2.PT := T#0MS;
   S703_TL_DC_2ND_CLAMP2.Error_T2.Q := FALSE;
   S703_TL_DC_2ND_CLAMP2.Error_T2.ET := T#0MS;
   S703_TL_DC_2ND_CLAMP2.Error_T2.STATE := B#16#0;
   S703_TL_DC_2ND_CLAMP2.Error_T2.STIME := T#0MS;
   S703_TL_DC_2ND_CLAMP2.Error_T2.ATIME := T#0MS;
   S703_TL_DC_2ND_CLAMP2.Adv_End_Aux := FALSE;
   S703_TL_DC_2ND_CLAMP2.Ret_End_Aux := FALSE;
   S703_TL_DC_2ND_CLAMP2.CHK_Aux1 := FALSE;
   S703_TL_DC_2ND_CLAMP2.CHK_Aux2 := FALSE;
   S703_TL_DC_2ND_CLAMP2.Error_T1_DN := FALSE;
   S703_TL_DC_2ND_CLAMP2.Error_T2_DN := FALSE;
   S703_TL_DC_2ND_CLAMP2.Adv_Memo := FALSE;
   S703_TL_DC_2ND_CLAMP2.Visu_Adv_Arr[0] := FALSE;
   S703_TL_DC_2ND_CLAMP2.Visu_Adv_Arr[1] := FALSE;
   S703_TL_DC_2ND_CLAMP2.Visu_Adv_Arr[2] := FALSE;
   S703_TL_DC_2ND_CLAMP2.Visu_Adv_Arr[3] := FALSE;
   S703_TL_DC_2ND_CLAMP2.Visu_Adv_Arr[4] := FALSE;
   S703_TL_DC_2ND_CLAMP2.Visu_Adv_Arr[5] := FALSE;
   S703_TL_DC_2ND_CLAMP2.Visu_Adv_Arr[6] := FALSE;
   S703_TL_DC_2ND_CLAMP2.Visu_Adv_Arr[7] := FALSE;
   S703_TL_DC_2ND_CLAMP2.Visu_Adv_Arr[8] := FALSE;
   S703_TL_DC_2ND_CLAMP2.Visu_Adv_Arr[9] := FALSE;
   S703_TL_DC_2ND_CLAMP2.Visu_Adv_Arr[10] := FALSE;
   S703_TL_DC_2ND_CLAMP2.Visu_Adv_Arr[11] := FALSE;
   S703_TL_DC_2ND_CLAMP2.Visu_Adv_Arr[12] := FALSE;
   S703_TL_DC_2ND_CLAMP2.Visu_Adv_Arr[13] := FALSE;
   S703_TL_DC_2ND_CLAMP2.Visu_Adv_Arr[14] := FALSE;
   S703_TL_DC_2ND_CLAMP2.Visu_Adv_Arr[15] := FALSE;
   S703_TL_DC_2ND_CLAMP2.Visu_Ret_Arr[0] := FALSE;
   S703_TL_DC_2ND_CLAMP2.Visu_Ret_Arr[1] := FALSE;
   S703_TL_DC_2ND_CLAMP2.Visu_Ret_Arr[2] := FALSE;
   S703_TL_DC_2ND_CLAMP2.Visu_Ret_Arr[3] := FALSE;
   S703_TL_DC_2ND_CLAMP2.Visu_Ret_Arr[4] := FALSE;
   S703_TL_DC_2ND_CLAMP2.Visu_Ret_Arr[5] := FALSE;
   S703_TL_DC_2ND_CLAMP2.Visu_Ret_Arr[6] := FALSE;
   S703_TL_DC_2ND_CLAMP2.Visu_Ret_Arr[7] := FALSE;
   S703_TL_DC_2ND_CLAMP2.Visu_Ret_Arr[8] := FALSE;
   S703_TL_DC_2ND_CLAMP2.Visu_Ret_Arr[9] := FALSE;
   S703_TL_DC_2ND_CLAMP2.Visu_Ret_Arr[10] := FALSE;
   S703_TL_DC_2ND_CLAMP2.Visu_Ret_Arr[11] := FALSE;
   S703_TL_DC_2ND_CLAMP2.Visu_Ret_Arr[12] := FALSE;
   S703_TL_DC_2ND_CLAMP2.Visu_Ret_Arr[13] := FALSE;
   S703_TL_DC_2ND_CLAMP2.Visu_Ret_Arr[14] := FALSE;
   S703_TL_DC_2ND_CLAMP2.Visu_Ret_Arr[15] := FALSE;
   S703_TL_DC_2ND_CLAMP2.BLK_Move_Ret := 0;
   S703_TL_DC_2ND_CLAMP2.Enable := FALSE;
   S703_TL_DC_2ND_CLAMP2.Adv_End := FALSE;
   S703_TL_DC_2ND_CLAMP2.Ret_End := FALSE;
   S703_TL_DC_U261.Enable_Aux := FALSE;
   S703_TL_DC_U261.Adv_Amount := 0;
   S703_TL_DC_U261.Ret_Amount := 0;
   S703_TL_DC_U261.LS_Adv1 := FALSE;
   S703_TL_DC_U261.LS_Ret1 := FALSE;
   S703_TL_DC_U261.LS_Adv2 := FALSE;
   S703_TL_DC_U261.LS_Ret2 := FALSE;
   S703_TL_DC_U261.LS_Adv3 := FALSE;
   S703_TL_DC_U261.LS_Ret3 := FALSE;
   S703_TL_DC_U261.LS_Adv4 := FALSE;
   S703_TL_DC_U261.LS_Ret4 := FALSE;
   S703_TL_DC_U261.LS_Adv5 := FALSE;
   S703_TL_DC_U261.LS_Ret5 := FALSE;
   S703_TL_DC_U261.LS_Adv6 := FALSE;
   S703_TL_DC_U261.LS_Ret6 := FALSE;
   S703_TL_DC_U261.LS_Adv7 := FALSE;
   S703_TL_DC_U261.LS_Ret7 := FALSE;
   S703_TL_DC_U261.LS_Adv8 := FALSE;
   S703_TL_DC_U261.LS_Ret8 := FALSE;
   S703_TL_DC_U261.SOL_Adv := FALSE;
   S703_TL_DC_U261.SOL_Ret := FALSE;
   S703_TL_DC_U261.M_Ready := FALSE;
   S703_TL_DC_U261.T_CHK1 := T#0MS;
   S703_TL_DC_U261.T_CHK2 := T#0MS;
   S703_TL_DC_U261.PB_Lamp_CHK := FALSE;
   S703_TL_DC_U261.PB_Error_Rst := FALSE;
   S703_TL_DC_U261.M_FLICK := FALSE;
   S703_TL_DC_U261.M_Adv_Err := FALSE;
   S703_TL_DC_U261.M_Ret_Err := FALSE;
   S703_TL_DC_U261.LP_Adv := FALSE;
   S703_TL_DC_U261.LP_Ret := FALSE;
   S703_TL_DC_U261.Visu_Adv := W#16#0;
   S703_TL_DC_U261.Visu_Ret := W#16#0;
   S703_TL_DC_U261.Error_T1.IN := FALSE;
   S703_TL_DC_U261.Error_T1.PT := T#0MS;
   S703_TL_DC_U261.Error_T1.Q := FALSE;
   S703_TL_DC_U261.Error_T1.ET := T#0MS;
   S703_TL_DC_U261.Error_T1.STATE := B#16#0;
   S703_TL_DC_U261.Error_T1.STIME := T#0MS;
   S703_TL_DC_U261.Error_T1.ATIME := T#0MS;
   S703_TL_DC_U261.Error_T2.IN := FALSE;
   S703_TL_DC_U261.Error_T2.PT := T#0MS;
   S703_TL_DC_U261.Error_T2.Q := FALSE;
   S703_TL_DC_U261.Error_T2.ET := T#0MS;
   S703_TL_DC_U261.Error_T2.STATE := B#16#0;
   S703_TL_DC_U261.Error_T2.STIME := T#0MS;
   S703_TL_DC_U261.Error_T2.ATIME := T#0MS;
   S703_TL_DC_U261.Adv_End_Aux := FALSE;
   S703_TL_DC_U261.Ret_End_Aux := FALSE;
   S703_TL_DC_U261.CHK_Aux1 := FALSE;
   S703_TL_DC_U261.CHK_Aux2 := FALSE;
   S703_TL_DC_U261.Error_T1_DN := FALSE;
   S703_TL_DC_U261.Error_T2_DN := FALSE;
   S703_TL_DC_U261.Adv_Memo := FALSE;
   S703_TL_DC_U261.Visu_Adv_Arr[0] := FALSE;
   S703_TL_DC_U261.Visu_Adv_Arr[1] := FALSE;
   S703_TL_DC_U261.Visu_Adv_Arr[2] := FALSE;
   S703_TL_DC_U261.Visu_Adv_Arr[3] := FALSE;
   S703_TL_DC_U261.Visu_Adv_Arr[4] := FALSE;
   S703_TL_DC_U261.Visu_Adv_Arr[5] := FALSE;
   S703_TL_DC_U261.Visu_Adv_Arr[6] := FALSE;
   S703_TL_DC_U261.Visu_Adv_Arr[7] := FALSE;
   S703_TL_DC_U261.Visu_Adv_Arr[8] := FALSE;
   S703_TL_DC_U261.Visu_Adv_Arr[9] := FALSE;
   S703_TL_DC_U261.Visu_Adv_Arr[10] := FALSE;
   S703_TL_DC_U261.Visu_Adv_Arr[11] := FALSE;
   S703_TL_DC_U261.Visu_Adv_Arr[12] := FALSE;
   S703_TL_DC_U261.Visu_Adv_Arr[13] := FALSE;
   S703_TL_DC_U261.Visu_Adv_Arr[14] := FALSE;
   S703_TL_DC_U261.Visu_Adv_Arr[15] := FALSE;
   S703_TL_DC_U261.Visu_Ret_Arr[0] := FALSE;
   S703_TL_DC_U261.Visu_Ret_Arr[1] := FALSE;
   S703_TL_DC_U261.Visu_Ret_Arr[2] := FALSE;
   S703_TL_DC_U261.Visu_Ret_Arr[3] := FALSE;
   S703_TL_DC_U261.Visu_Ret_Arr[4] := FALSE;
   S703_TL_DC_U261.Visu_Ret_Arr[5] := FALSE;
   S703_TL_DC_U261.Visu_Ret_Arr[6] := FALSE;
   S703_TL_DC_U261.Visu_Ret_Arr[7] := FALSE;
   S703_TL_DC_U261.Visu_Ret_Arr[8] := FALSE;
   S703_TL_DC_U261.Visu_Ret_Arr[9] := FALSE;
   S703_TL_DC_U261.Visu_Ret_Arr[10] := FALSE;
   S703_TL_DC_U261.Visu_Ret_Arr[11] := FALSE;
   S703_TL_DC_U261.Visu_Ret_Arr[12] := FALSE;
   S703_TL_DC_U261.Visu_Ret_Arr[13] := FALSE;
   S703_TL_DC_U261.Visu_Ret_Arr[14] := FALSE;
   S703_TL_DC_U261.Visu_Ret_Arr[15] := FALSE;
   S703_TL_DC_U261.BLK_Move_Ret := 0;
   S703_TL_DC_U261.Enable := FALSE;
   S703_TL_DC_U261.Adv_End := FALSE;
   S703_TL_DC_U261.Ret_End := FALSE;
   S703_TL_DC_U261_CLAMP.Enable_Aux := FALSE;
   S703_TL_DC_U261_CLAMP.Adv_Amount := 0;
   S703_TL_DC_U261_CLAMP.Ret_Amount := 0;
   S703_TL_DC_U261_CLAMP.LS_Adv1 := FALSE;
   S703_TL_DC_U261_CLAMP.LS_Ret1 := FALSE;
   S703_TL_DC_U261_CLAMP.LS_Adv2 := FALSE;
   S703_TL_DC_U261_CLAMP.LS_Ret2 := FALSE;
   S703_TL_DC_U261_CLAMP.LS_Adv3 := FALSE;
   S703_TL_DC_U261_CLAMP.LS_Ret3 := FALSE;
   S703_TL_DC_U261_CLAMP.LS_Adv4 := FALSE;
   S703_TL_DC_U261_CLAMP.LS_Ret4 := FALSE;
   S703_TL_DC_U261_CLAMP.LS_Adv5 := FALSE;
   S703_TL_DC_U261_CLAMP.LS_Ret5 := FALSE;
   S703_TL_DC_U261_CLAMP.LS_Adv6 := FALSE;
   S703_TL_DC_U261_CLAMP.LS_Ret6 := FALSE;
   S703_TL_DC_U261_CLAMP.LS_Adv7 := FALSE;
   S703_TL_DC_U261_CLAMP.LS_Ret7 := FALSE;
   S703_TL_DC_U261_CLAMP.LS_Adv8 := FALSE;
   S703_TL_DC_U261_CLAMP.LS_Ret8 := FALSE;
   S703_TL_DC_U261_CLAMP.SOL_Adv := FALSE;
   S703_TL_DC_U261_CLAMP.SOL_Ret := FALSE;
   S703_TL_DC_U261_CLAMP.M_Ready := FALSE;
   S703_TL_DC_U261_CLAMP.T_CHK1 := T#0MS;
   S703_TL_DC_U261_CLAMP.T_CHK2 := T#0MS;
   S703_TL_DC_U261_CLAMP.PB_Lamp_CHK := FALSE;
   S703_TL_DC_U261_CLAMP.PB_Error_Rst := FALSE;
   S703_TL_DC_U261_CLAMP.M_FLICK := FALSE;
   S703_TL_DC_U261_CLAMP.M_Adv_Err := FALSE;
   S703_TL_DC_U261_CLAMP.M_Ret_Err := FALSE;
   S703_TL_DC_U261_CLAMP.LP_Adv := FALSE;
   S703_TL_DC_U261_CLAMP.LP_Ret := FALSE;
   S703_TL_DC_U261_CLAMP.Visu_Adv := W#16#0;
   S703_TL_DC_U261_CLAMP.Visu_Ret := W#16#0;
   S703_TL_DC_U261_CLAMP.Error_T1.IN := FALSE;
   S703_TL_DC_U261_CLAMP.Error_T1.PT := T#0MS;
   S703_TL_DC_U261_CLAMP.Error_T1.Q := FALSE;
   S703_TL_DC_U261_CLAMP.Error_T1.ET := T#0MS;
   S703_TL_DC_U261_CLAMP.Error_T1.STATE := B#16#0;
   S703_TL_DC_U261_CLAMP.Error_T1.STIME := T#0MS;
   S703_TL_DC_U261_CLAMP.Error_T1.ATIME := T#0MS;
   S703_TL_DC_U261_CLAMP.Error_T2.IN := FALSE;
   S703_TL_DC_U261_CLAMP.Error_T2.PT := T#0MS;
   S703_TL_DC_U261_CLAMP.Error_T2.Q := FALSE;
   S703_TL_DC_U261_CLAMP.Error_T2.ET := T#0MS;
   S703_TL_DC_U261_CLAMP.Error_T2.STATE := B#16#0;
   S703_TL_DC_U261_CLAMP.Error_T2.STIME := T#0MS;
   S703_TL_DC_U261_CLAMP.Error_T2.ATIME := T#0MS;
   S703_TL_DC_U261_CLAMP.Adv_End_Aux := FALSE;
   S703_TL_DC_U261_CLAMP.Ret_End_Aux := FALSE;
   S703_TL_DC_U261_CLAMP.CHK_Aux1 := FALSE;
   S703_TL_DC_U261_CLAMP.CHK_Aux2 := FALSE;
   S703_TL_DC_U261_CLAMP.Error_T1_DN := FALSE;
   S703_TL_DC_U261_CLAMP.Error_T2_DN := FALSE;
   S703_TL_DC_U261_CLAMP.Adv_Memo := FALSE;
   S703_TL_DC_U261_CLAMP.Visu_Adv_Arr[0] := FALSE;
   S703_TL_DC_U261_CLAMP.Visu_Adv_Arr[1] := FALSE;
   S703_TL_DC_U261_CLAMP.Visu_Adv_Arr[2] := FALSE;
   S703_TL_DC_U261_CLAMP.Visu_Adv_Arr[3] := FALSE;
   S703_TL_DC_U261_CLAMP.Visu_Adv_Arr[4] := FALSE;
   S703_TL_DC_U261_CLAMP.Visu_Adv_Arr[5] := FALSE;
   S703_TL_DC_U261_CLAMP.Visu_Adv_Arr[6] := FALSE;
   S703_TL_DC_U261_CLAMP.Visu_Adv_Arr[7] := FALSE;
   S703_TL_DC_U261_CLAMP.Visu_Adv_Arr[8] := FALSE;
   S703_TL_DC_U261_CLAMP.Visu_Adv_Arr[9] := FALSE;
   S703_TL_DC_U261_CLAMP.Visu_Adv_Arr[10] := FALSE;
   S703_TL_DC_U261_CLAMP.Visu_Adv_Arr[11] := FALSE;
   S703_TL_DC_U261_CLAMP.Visu_Adv_Arr[12] := FALSE;
   S703_TL_DC_U261_CLAMP.Visu_Adv_Arr[13] := FALSE;
   S703_TL_DC_U261_CLAMP.Visu_Adv_Arr[14] := FALSE;
   S703_TL_DC_U261_CLAMP.Visu_Adv_Arr[15] := FALSE;
   S703_TL_DC_U261_CLAMP.Visu_Ret_Arr[0] := FALSE;
   S703_TL_DC_U261_CLAMP.Visu_Ret_Arr[1] := FALSE;
   S703_TL_DC_U261_CLAMP.Visu_Ret_Arr[2] := FALSE;
   S703_TL_DC_U261_CLAMP.Visu_Ret_Arr[3] := FALSE;
   S703_TL_DC_U261_CLAMP.Visu_Ret_Arr[4] := FALSE;
   S703_TL_DC_U261_CLAMP.Visu_Ret_Arr[5] := FALSE;
   S703_TL_DC_U261_CLAMP.Visu_Ret_Arr[6] := FALSE;
   S703_TL_DC_U261_CLAMP.Visu_Ret_Arr[7] := FALSE;
   S703_TL_DC_U261_CLAMP.Visu_Ret_Arr[8] := FALSE;
   S703_TL_DC_U261_CLAMP.Visu_Ret_Arr[9] := FALSE;
   S703_TL_DC_U261_CLAMP.Visu_Ret_Arr[10] := FALSE;
   S703_TL_DC_U261_CLAMP.Visu_Ret_Arr[11] := FALSE;
   S703_TL_DC_U261_CLAMP.Visu_Ret_Arr[12] := FALSE;
   S703_TL_DC_U261_CLAMP.Visu_Ret_Arr[13] := FALSE;
   S703_TL_DC_U261_CLAMP.Visu_Ret_Arr[14] := FALSE;
   S703_TL_DC_U261_CLAMP.Visu_Ret_Arr[15] := FALSE;
   S703_TL_DC_U261_CLAMP.BLK_Move_Ret := 0;
   S703_TL_DC_U261_CLAMP.Enable := FALSE;
   S703_TL_DC_U261_CLAMP.Adv_End := FALSE;
   S703_TL_DC_U261_CLAMP.Ret_End := FALSE;
   S703_TL_DC_U269.Enable_Aux := FALSE;
   S703_TL_DC_U269.Adv_Amount := 0;
   S703_TL_DC_U269.Ret_Amount := 0;
   S703_TL_DC_U269.LS_Adv1 := FALSE;
   S703_TL_DC_U269.LS_Ret1 := FALSE;
   S703_TL_DC_U269.LS_Adv2 := FALSE;
   S703_TL_DC_U269.LS_Ret2 := FALSE;
   S703_TL_DC_U269.LS_Adv3 := FALSE;
   S703_TL_DC_U269.LS_Ret3 := FALSE;
   S703_TL_DC_U269.LS_Adv4 := FALSE;
   S703_TL_DC_U269.LS_Ret4 := FALSE;
   S703_TL_DC_U269.LS_Adv5 := FALSE;
   S703_TL_DC_U269.LS_Ret5 := FALSE;
   S703_TL_DC_U269.LS_Adv6 := FALSE;
   S703_TL_DC_U269.LS_Ret6 := FALSE;
   S703_TL_DC_U269.LS_Adv7 := FALSE;
   S703_TL_DC_U269.LS_Ret7 := FALSE;
   S703_TL_DC_U269.LS_Adv8 := FALSE;
   S703_TL_DC_U269.LS_Ret8 := FALSE;
   S703_TL_DC_U269.SOL_Adv := FALSE;
   S703_TL_DC_U269.SOL_Ret := FALSE;
   S703_TL_DC_U269.M_Ready := FALSE;
   S703_TL_DC_U269.T_CHK1 := T#0MS;
   S703_TL_DC_U269.T_CHK2 := T#0MS;
   S703_TL_DC_U269.PB_Lamp_CHK := FALSE;
   S703_TL_DC_U269.PB_Error_Rst := FALSE;
   S703_TL_DC_U269.M_FLICK := FALSE;
   S703_TL_DC_U269.M_Adv_Err := FALSE;
   S703_TL_DC_U269.M_Ret_Err := FALSE;
   S703_TL_DC_U269.LP_Adv := FALSE;
   S703_TL_DC_U269.LP_Ret := FALSE;
   S703_TL_DC_U269.Visu_Adv := W#16#0;
   S703_TL_DC_U269.Visu_Ret := W#16#0;
   S703_TL_DC_U269.Error_T1.IN := FALSE;
   S703_TL_DC_U269.Error_T1.PT := T#0MS;
   S703_TL_DC_U269.Error_T1.Q := FALSE;
   S703_TL_DC_U269.Error_T1.ET := T#0MS;
   S703_TL_DC_U269.Error_T1.STATE := B#16#0;
   S703_TL_DC_U269.Error_T1.STIME := T#0MS;
   S703_TL_DC_U269.Error_T1.ATIME := T#0MS;
   S703_TL_DC_U269.Error_T2.IN := FALSE;
   S703_TL_DC_U269.Error_T2.PT := T#0MS;
   S703_TL_DC_U269.Error_T2.Q := FALSE;
   S703_TL_DC_U269.Error_T2.ET := T#0MS;
   S703_TL_DC_U269.Error_T2.STATE := B#16#0;
   S703_TL_DC_U269.Error_T2.STIME := T#0MS;
   S703_TL_DC_U269.Error_T2.ATIME := T#0MS;
   S703_TL_DC_U269.Adv_End_Aux := FALSE;
   S703_TL_DC_U269.Ret_End_Aux := FALSE;
   S703_TL_DC_U269.CHK_Aux1 := FALSE;
   S703_TL_DC_U269.CHK_Aux2 := FALSE;
   S703_TL_DC_U269.Error_T1_DN := FALSE;
   S703_TL_DC_U269.Error_T2_DN := FALSE;
   S703_TL_DC_U269.Adv_Memo := FALSE;
   S703_TL_DC_U269.Visu_Adv_Arr[0] := FALSE;
   S703_TL_DC_U269.Visu_Adv_Arr[1] := FALSE;
   S703_TL_DC_U269.Visu_Adv_Arr[2] := FALSE;
   S703_TL_DC_U269.Visu_Adv_Arr[3] := FALSE;
   S703_TL_DC_U269.Visu_Adv_Arr[4] := FALSE;
   S703_TL_DC_U269.Visu_Adv_Arr[5] := FALSE;
   S703_TL_DC_U269.Visu_Adv_Arr[6] := FALSE;
   S703_TL_DC_U269.Visu_Adv_Arr[7] := FALSE;
   S703_TL_DC_U269.Visu_Adv_Arr[8] := FALSE;
   S703_TL_DC_U269.Visu_Adv_Arr[9] := FALSE;
   S703_TL_DC_U269.Visu_Adv_Arr[10] := FALSE;
   S703_TL_DC_U269.Visu_Adv_Arr[11] := FALSE;
   S703_TL_DC_U269.Visu_Adv_Arr[12] := FALSE;
   S703_TL_DC_U269.Visu_Adv_Arr[13] := FALSE;
   S703_TL_DC_U269.Visu_Adv_Arr[14] := FALSE;
   S703_TL_DC_U269.Visu_Adv_Arr[15] := FALSE;
   S703_TL_DC_U269.Visu_Ret_Arr[0] := FALSE;
   S703_TL_DC_U269.Visu_Ret_Arr[1] := FALSE;
   S703_TL_DC_U269.Visu_Ret_Arr[2] := FALSE;
   S703_TL_DC_U269.Visu_Ret_Arr[3] := FALSE;
   S703_TL_DC_U269.Visu_Ret_Arr[4] := FALSE;
   S703_TL_DC_U269.Visu_Ret_Arr[5] := FALSE;
   S703_TL_DC_U269.Visu_Ret_Arr[6] := FALSE;
   S703_TL_DC_U269.Visu_Ret_Arr[7] := FALSE;
   S703_TL_DC_U269.Visu_Ret_Arr[8] := FALSE;
   S703_TL_DC_U269.Visu_Ret_Arr[9] := FALSE;
   S703_TL_DC_U269.Visu_Ret_Arr[10] := FALSE;
   S703_TL_DC_U269.Visu_Ret_Arr[11] := FALSE;
   S703_TL_DC_U269.Visu_Ret_Arr[12] := FALSE;
   S703_TL_DC_U269.Visu_Ret_Arr[13] := FALSE;
   S703_TL_DC_U269.Visu_Ret_Arr[14] := FALSE;
   S703_TL_DC_U269.Visu_Ret_Arr[15] := FALSE;
   S703_TL_DC_U269.BLK_Move_Ret := 0;
   S703_TL_DC_U269.Enable := FALSE;
   S703_TL_DC_U269.Adv_End := FALSE;
   S703_TL_DC_U269.Ret_End := FALSE;
   S703_TL_DC_U269_CLAMP.Enable_Aux := FALSE;
   S703_TL_DC_U269_CLAMP.Adv_Amount := 0;
   S703_TL_DC_U269_CLAMP.Ret_Amount := 0;
   S703_TL_DC_U269_CLAMP.LS_Adv1 := FALSE;
   S703_TL_DC_U269_CLAMP.LS_Ret1 := FALSE;
   S703_TL_DC_U269_CLAMP.LS_Adv2 := FALSE;
   S703_TL_DC_U269_CLAMP.LS_Ret2 := FALSE;
   S703_TL_DC_U269_CLAMP.LS_Adv3 := FALSE;
   S703_TL_DC_U269_CLAMP.LS_Ret3 := FALSE;
   S703_TL_DC_U269_CLAMP.LS_Adv4 := FALSE;
   S703_TL_DC_U269_CLAMP.LS_Ret4 := FALSE;
   S703_TL_DC_U269_CLAMP.LS_Adv5 := FALSE;
   S703_TL_DC_U269_CLAMP.LS_Ret5 := FALSE;
   S703_TL_DC_U269_CLAMP.LS_Adv6 := FALSE;
   S703_TL_DC_U269_CLAMP.LS_Ret6 := FALSE;
   S703_TL_DC_U269_CLAMP.LS_Adv7 := FALSE;
   S703_TL_DC_U269_CLAMP.LS_Ret7 := FALSE;
   S703_TL_DC_U269_CLAMP.LS_Adv8 := FALSE;
   S703_TL_DC_U269_CLAMP.LS_Ret8 := FALSE;
   S703_TL_DC_U269_CLAMP.SOL_Adv := FALSE;
   S703_TL_DC_U269_CLAMP.SOL_Ret := FALSE;
   S703_TL_DC_U269_CLAMP.M_Ready := FALSE;
   S703_TL_DC_U269_CLAMP.T_CHK1 := T#0MS;
   S703_TL_DC_U269_CLAMP.T_CHK2 := T#0MS;
   S703_TL_DC_U269_CLAMP.PB_Lamp_CHK := FALSE;
   S703_TL_DC_U269_CLAMP.PB_Error_Rst := FALSE;
   S703_TL_DC_U269_CLAMP.M_FLICK := FALSE;
   S703_TL_DC_U269_CLAMP.M_Adv_Err := FALSE;
   S703_TL_DC_U269_CLAMP.M_Ret_Err := FALSE;
   S703_TL_DC_U269_CLAMP.LP_Adv := FALSE;
   S703_TL_DC_U269_CLAMP.LP_Ret := FALSE;
   S703_TL_DC_U269_CLAMP.Visu_Adv := W#16#0;
   S703_TL_DC_U269_CLAMP.Visu_Ret := W#16#0;
   S703_TL_DC_U269_CLAMP.Error_T1.IN := FALSE;
   S703_TL_DC_U269_CLAMP.Error_T1.PT := T#0MS;
   S703_TL_DC_U269_CLAMP.Error_T1.Q := FALSE;
   S703_TL_DC_U269_CLAMP.Error_T1.ET := T#0MS;
   S703_TL_DC_U269_CLAMP.Error_T1.STATE := B#16#0;
   S703_TL_DC_U269_CLAMP.Error_T1.STIME := T#0MS;
   S703_TL_DC_U269_CLAMP.Error_T1.ATIME := T#0MS;
   S703_TL_DC_U269_CLAMP.Error_T2.IN := FALSE;
   S703_TL_DC_U269_CLAMP.Error_T2.PT := T#0MS;
   S703_TL_DC_U269_CLAMP.Error_T2.Q := FALSE;
   S703_TL_DC_U269_CLAMP.Error_T2.ET := T#0MS;
   S703_TL_DC_U269_CLAMP.Error_T2.STATE := B#16#0;
   S703_TL_DC_U269_CLAMP.Error_T2.STIME := T#0MS;
   S703_TL_DC_U269_CLAMP.Error_T2.ATIME := T#0MS;
   S703_TL_DC_U269_CLAMP.Adv_End_Aux := FALSE;
   S703_TL_DC_U269_CLAMP.Ret_End_Aux := FALSE;
   S703_TL_DC_U269_CLAMP.CHK_Aux1 := FALSE;
   S703_TL_DC_U269_CLAMP.CHK_Aux2 := FALSE;
   S703_TL_DC_U269_CLAMP.Error_T1_DN := FALSE;
   S703_TL_DC_U269_CLAMP.Error_T2_DN := FALSE;
   S703_TL_DC_U269_CLAMP.Adv_Memo := FALSE;
   S703_TL_DC_U269_CLAMP.Visu_Adv_Arr[0] := FALSE;
   S703_TL_DC_U269_CLAMP.Visu_Adv_Arr[1] := FALSE;
   S703_TL_DC_U269_CLAMP.Visu_Adv_Arr[2] := FALSE;
   S703_TL_DC_U269_CLAMP.Visu_Adv_Arr[3] := FALSE;
   S703_TL_DC_U269_CLAMP.Visu_Adv_Arr[4] := FALSE;
   S703_TL_DC_U269_CLAMP.Visu_Adv_Arr[5] := FALSE;
   S703_TL_DC_U269_CLAMP.Visu_Adv_Arr[6] := FALSE;
   S703_TL_DC_U269_CLAMP.Visu_Adv_Arr[7] := FALSE;
   S703_TL_DC_U269_CLAMP.Visu_Adv_Arr[8] := FALSE;
   S703_TL_DC_U269_CLAMP.Visu_Adv_Arr[9] := FALSE;
   S703_TL_DC_U269_CLAMP.Visu_Adv_Arr[10] := FALSE;
   S703_TL_DC_U269_CLAMP.Visu_Adv_Arr[11] := FALSE;
   S703_TL_DC_U269_CLAMP.Visu_Adv_Arr[12] := FALSE;
   S703_TL_DC_U269_CLAMP.Visu_Adv_Arr[13] := FALSE;
   S703_TL_DC_U269_CLAMP.Visu_Adv_Arr[14] := FALSE;
   S703_TL_DC_U269_CLAMP.Visu_Adv_Arr[15] := FALSE;
   S703_TL_DC_U269_CLAMP.Visu_Ret_Arr[0] := FALSE;
   S703_TL_DC_U269_CLAMP.Visu_Ret_Arr[1] := FALSE;
   S703_TL_DC_U269_CLAMP.Visu_Ret_Arr[2] := FALSE;
   S703_TL_DC_U269_CLAMP.Visu_Ret_Arr[3] := FALSE;
   S703_TL_DC_U269_CLAMP.Visu_Ret_Arr[4] := FALSE;
   S703_TL_DC_U269_CLAMP.Visu_Ret_Arr[5] := FALSE;
   S703_TL_DC_U269_CLAMP.Visu_Ret_Arr[6] := FALSE;
   S703_TL_DC_U269_CLAMP.Visu_Ret_Arr[7] := FALSE;
   S703_TL_DC_U269_CLAMP.Visu_Ret_Arr[8] := FALSE;
   S703_TL_DC_U269_CLAMP.Visu_Ret_Arr[9] := FALSE;
   S703_TL_DC_U269_CLAMP.Visu_Ret_Arr[10] := FALSE;
   S703_TL_DC_U269_CLAMP.Visu_Ret_Arr[11] := FALSE;
   S703_TL_DC_U269_CLAMP.Visu_Ret_Arr[12] := FALSE;
   S703_TL_DC_U269_CLAMP.Visu_Ret_Arr[13] := FALSE;
   S703_TL_DC_U269_CLAMP.Visu_Ret_Arr[14] := FALSE;
   S703_TL_DC_U269_CLAMP.Visu_Ret_Arr[15] := FALSE;
   S703_TL_DC_U269_CLAMP.BLK_Move_Ret := 0;
   S703_TL_DC_U269_CLAMP.Enable := FALSE;
   S703_TL_DC_U269_CLAMP.Adv_End := FALSE;
   S703_TL_DC_U269_CLAMP.Ret_End := FALSE;
   S703_TL_DC_3RD_CLAMP.Enable_Aux := FALSE;
   S703_TL_DC_3RD_CLAMP.Adv_Amount := 0;
   S703_TL_DC_3RD_CLAMP.Ret_Amount := 0;
   S703_TL_DC_3RD_CLAMP.LS_Adv1 := FALSE;
   S703_TL_DC_3RD_CLAMP.LS_Ret1 := FALSE;
   S703_TL_DC_3RD_CLAMP.LS_Adv2 := FALSE;
   S703_TL_DC_3RD_CLAMP.LS_Ret2 := FALSE;
   S703_TL_DC_3RD_CLAMP.LS_Adv3 := FALSE;
   S703_TL_DC_3RD_CLAMP.LS_Ret3 := FALSE;
   S703_TL_DC_3RD_CLAMP.LS_Adv4 := FALSE;
   S703_TL_DC_3RD_CLAMP.LS_Ret4 := FALSE;
   S703_TL_DC_3RD_CLAMP.LS_Adv5 := FALSE;
   S703_TL_DC_3RD_CLAMP.LS_Ret5 := FALSE;
   S703_TL_DC_3RD_CLAMP.LS_Adv6 := FALSE;
   S703_TL_DC_3RD_CLAMP.LS_Ret6 := FALSE;
   S703_TL_DC_3RD_CLAMP.LS_Adv7 := FALSE;
   S703_TL_DC_3RD_CLAMP.LS_Ret7 := FALSE;
   S703_TL_DC_3RD_CLAMP.LS_Adv8 := FALSE;
   S703_TL_DC_3RD_CLAMP.LS_Ret8 := FALSE;
   S703_TL_DC_3RD_CLAMP.SOL_Adv := FALSE;
   S703_TL_DC_3RD_CLAMP.SOL_Ret := FALSE;
   S703_TL_DC_3RD_CLAMP.M_Ready := FALSE;
   S703_TL_DC_3RD_CLAMP.T_CHK1 := T#0MS;
   S703_TL_DC_3RD_CLAMP.T_CHK2 := T#0MS;
   S703_TL_DC_3RD_CLAMP.PB_Lamp_CHK := FALSE;
   S703_TL_DC_3RD_CLAMP.PB_Error_Rst := FALSE;
   S703_TL_DC_3RD_CLAMP.M_FLICK := FALSE;
   S703_TL_DC_3RD_CLAMP.M_Adv_Err := FALSE;
   S703_TL_DC_3RD_CLAMP.M_Ret_Err := FALSE;
   S703_TL_DC_3RD_CLAMP.LP_Adv := FALSE;
   S703_TL_DC_3RD_CLAMP.LP_Ret := FALSE;
   S703_TL_DC_3RD_CLAMP.Visu_Adv := W#16#0;
   S703_TL_DC_3RD_CLAMP.Visu_Ret := W#16#0;
   S703_TL_DC_3RD_CLAMP.Error_T1.IN := FALSE;
   S703_TL_DC_3RD_CLAMP.Error_T1.PT := T#0MS;
   S703_TL_DC_3RD_CLAMP.Error_T1.Q := FALSE;
   S703_TL_DC_3RD_CLAMP.Error_T1.ET := T#0MS;
   S703_TL_DC_3RD_CLAMP.Error_T1.STATE := B#16#0;
   S703_TL_DC_3RD_CLAMP.Error_T1.STIME := T#0MS;
   S703_TL_DC_3RD_CLAMP.Error_T1.ATIME := T#0MS;
   S703_TL_DC_3RD_CLAMP.Error_T2.IN := FALSE;
   S703_TL_DC_3RD_CLAMP.Error_T2.PT := T#0MS;
   S703_TL_DC_3RD_CLAMP.Error_T2.Q := FALSE;
   S703_TL_DC_3RD_CLAMP.Error_T2.ET := T#0MS;
   S703_TL_DC_3RD_CLAMP.Error_T2.STATE := B#16#0;
   S703_TL_DC_3RD_CLAMP.Error_T2.STIME := T#0MS;
   S703_TL_DC_3RD_CLAMP.Error_T2.ATIME := T#0MS;
   S703_TL_DC_3RD_CLAMP.Adv_End_Aux := FALSE;
   S703_TL_DC_3RD_CLAMP.Ret_End_Aux := FALSE;
   S703_TL_DC_3RD_CLAMP.CHK_Aux1 := FALSE;
   S703_TL_DC_3RD_CLAMP.CHK_Aux2 := FALSE;
   S703_TL_DC_3RD_CLAMP.Error_T1_DN := FALSE;
   S703_TL_DC_3RD_CLAMP.Error_T2_DN := FALSE;
   S703_TL_DC_3RD_CLAMP.Adv_Memo := FALSE;
   S703_TL_DC_3RD_CLAMP.Visu_Adv_Arr[0] := FALSE;
   S703_TL_DC_3RD_CLAMP.Visu_Adv_Arr[1] := FALSE;
   S703_TL_DC_3RD_CLAMP.Visu_Adv_Arr[2] := FALSE;
   S703_TL_DC_3RD_CLAMP.Visu_Adv_Arr[3] := FALSE;
   S703_TL_DC_3RD_CLAMP.Visu_Adv_Arr[4] := FALSE;
   S703_TL_DC_3RD_CLAMP.Visu_Adv_Arr[5] := FALSE;
   S703_TL_DC_3RD_CLAMP.Visu_Adv_Arr[6] := FALSE;
   S703_TL_DC_3RD_CLAMP.Visu_Adv_Arr[7] := FALSE;
   S703_TL_DC_3RD_CLAMP.Visu_Adv_Arr[8] := FALSE;
   S703_TL_DC_3RD_CLAMP.Visu_Adv_Arr[9] := FALSE;
   S703_TL_DC_3RD_CLAMP.Visu_Adv_Arr[10] := FALSE;
   S703_TL_DC_3RD_CLAMP.Visu_Adv_Arr[11] := FALSE;
   S703_TL_DC_3RD_CLAMP.Visu_Adv_Arr[12] := FALSE;
   S703_TL_DC_3RD_CLAMP.Visu_Adv_Arr[13] := FALSE;
   S703_TL_DC_3RD_CLAMP.Visu_Adv_Arr[14] := FALSE;
   S703_TL_DC_3RD_CLAMP.Visu_Adv_Arr[15] := FALSE;
   S703_TL_DC_3RD_CLAMP.Visu_Ret_Arr[0] := FALSE;
   S703_TL_DC_3RD_CLAMP.Visu_Ret_Arr[1] := FALSE;
   S703_TL_DC_3RD_CLAMP.Visu_Ret_Arr[2] := FALSE;
   S703_TL_DC_3RD_CLAMP.Visu_Ret_Arr[3] := FALSE;
   S703_TL_DC_3RD_CLAMP.Visu_Ret_Arr[4] := FALSE;
   S703_TL_DC_3RD_CLAMP.Visu_Ret_Arr[5] := FALSE;
   S703_TL_DC_3RD_CLAMP.Visu_Ret_Arr[6] := FALSE;
   S703_TL_DC_3RD_CLAMP.Visu_Ret_Arr[7] := FALSE;
   S703_TL_DC_3RD_CLAMP.Visu_Ret_Arr[8] := FALSE;
   S703_TL_DC_3RD_CLAMP.Visu_Ret_Arr[9] := FALSE;
   S703_TL_DC_3RD_CLAMP.Visu_Ret_Arr[10] := FALSE;
   S703_TL_DC_3RD_CLAMP.Visu_Ret_Arr[11] := FALSE;
   S703_TL_DC_3RD_CLAMP.Visu_Ret_Arr[12] := FALSE;
   S703_TL_DC_3RD_CLAMP.Visu_Ret_Arr[13] := FALSE;
   S703_TL_DC_3RD_CLAMP.Visu_Ret_Arr[14] := FALSE;
   S703_TL_DC_3RD_CLAMP.Visu_Ret_Arr[15] := FALSE;
   S703_TL_DC_3RD_CLAMP.BLK_Move_Ret := 0;
   S703_TL_DC_3RD_CLAMP.Enable := FALSE;
   S703_TL_DC_3RD_CLAMP.Adv_End := FALSE;
   S703_TL_DC_3RD_CLAMP.Ret_End := FALSE;
   S703_TL_DC_U262_1_UP_DN.Enable_Aux := FALSE;
   S703_TL_DC_U262_1_UP_DN.Adv_Amount := 0;
   S703_TL_DC_U262_1_UP_DN.Ret_Amount := 0;
   S703_TL_DC_U262_1_UP_DN.LS_Adv1 := FALSE;
   S703_TL_DC_U262_1_UP_DN.LS_Ret1 := FALSE;
   S703_TL_DC_U262_1_UP_DN.LS_Adv2 := FALSE;
   S703_TL_DC_U262_1_UP_DN.LS_Ret2 := FALSE;
   S703_TL_DC_U262_1_UP_DN.LS_Adv3 := FALSE;
   S703_TL_DC_U262_1_UP_DN.LS_Ret3 := FALSE;
   S703_TL_DC_U262_1_UP_DN.LS_Adv4 := FALSE;
   S703_TL_DC_U262_1_UP_DN.LS_Ret4 := FALSE;
   S703_TL_DC_U262_1_UP_DN.LS_Adv5 := FALSE;
   S703_TL_DC_U262_1_UP_DN.LS_Ret5 := FALSE;
   S703_TL_DC_U262_1_UP_DN.LS_Adv6 := FALSE;
   S703_TL_DC_U262_1_UP_DN.LS_Ret6 := FALSE;
   S703_TL_DC_U262_1_UP_DN.LS_Adv7 := FALSE;
   S703_TL_DC_U262_1_UP_DN.LS_Ret7 := FALSE;
   S703_TL_DC_U262_1_UP_DN.LS_Adv8 := FALSE;
   S703_TL_DC_U262_1_UP_DN.LS_Ret8 := FALSE;
   S703_TL_DC_U262_1_UP_DN.SOL_Adv := FALSE;
   S703_TL_DC_U262_1_UP_DN.SOL_Ret := FALSE;
   S703_TL_DC_U262_1_UP_DN.M_Ready := FALSE;
   S703_TL_DC_U262_1_UP_DN.T_CHK1 := T#0MS;
   S703_TL_DC_U262_1_UP_DN.T_CHK2 := T#0MS;
   S703_TL_DC_U262_1_UP_DN.PB_Lamp_CHK := FALSE;
   S703_TL_DC_U262_1_UP_DN.PB_Error_Rst := FALSE;
   S703_TL_DC_U262_1_UP_DN.M_FLICK := FALSE;
   S703_TL_DC_U262_1_UP_DN.M_Adv_Err := FALSE;
   S703_TL_DC_U262_1_UP_DN.M_Ret_Err := FALSE;
   S703_TL_DC_U262_1_UP_DN.LP_Adv := FALSE;
   S703_TL_DC_U262_1_UP_DN.LP_Ret := FALSE;
   S703_TL_DC_U262_1_UP_DN.Visu_Adv := W#16#0;
   S703_TL_DC_U262_1_UP_DN.Visu_Ret := W#16#0;
   S703_TL_DC_U262_1_UP_DN.Error_T1.IN := FALSE;
   S703_TL_DC_U262_1_UP_DN.Error_T1.PT := T#0MS;
   S703_TL_DC_U262_1_UP_DN.Error_T1.Q := FALSE;
   S703_TL_DC_U262_1_UP_DN.Error_T1.ET := T#0MS;
   S703_TL_DC_U262_1_UP_DN.Error_T1.STATE := B#16#0;
   S703_TL_DC_U262_1_UP_DN.Error_T1.STIME := T#0MS;
   S703_TL_DC_U262_1_UP_DN.Error_T1.ATIME := T#0MS;
   S703_TL_DC_U262_1_UP_DN.Error_T2.IN := FALSE;
   S703_TL_DC_U262_1_UP_DN.Error_T2.PT := T#0MS;
   S703_TL_DC_U262_1_UP_DN.Error_T2.Q := FALSE;
   S703_TL_DC_U262_1_UP_DN.Error_T2.ET := T#0MS;
   S703_TL_DC_U262_1_UP_DN.Error_T2.STATE := B#16#0;
   S703_TL_DC_U262_1_UP_DN.Error_T2.STIME := T#0MS;
   S703_TL_DC_U262_1_UP_DN.Error_T2.ATIME := T#0MS;
   S703_TL_DC_U262_1_UP_DN.Adv_End_Aux := FALSE;
   S703_TL_DC_U262_1_UP_DN.Ret_End_Aux := FALSE;
   S703_TL_DC_U262_1_UP_DN.CHK_Aux1 := FALSE;
   S703_TL_DC_U262_1_UP_DN.CHK_Aux2 := FALSE;
   S703_TL_DC_U262_1_UP_DN.Error_T1_DN := FALSE;
   S703_TL_DC_U262_1_UP_DN.Error_T2_DN := FALSE;
   S703_TL_DC_U262_1_UP_DN.Adv_Memo := FALSE;
   S703_TL_DC_U262_1_UP_DN.Visu_Adv_Arr[0] := FALSE;
   S703_TL_DC_U262_1_UP_DN.Visu_Adv_Arr[1] := FALSE;
   S703_TL_DC_U262_1_UP_DN.Visu_Adv_Arr[2] := FALSE;
   S703_TL_DC_U262_1_UP_DN.Visu_Adv_Arr[3] := FALSE;
   S703_TL_DC_U262_1_UP_DN.Visu_Adv_Arr[4] := FALSE;
   S703_TL_DC_U262_1_UP_DN.Visu_Adv_Arr[5] := FALSE;
   S703_TL_DC_U262_1_UP_DN.Visu_Adv_Arr[6] := FALSE;
   S703_TL_DC_U262_1_UP_DN.Visu_Adv_Arr[7] := FALSE;
   S703_TL_DC_U262_1_UP_DN.Visu_Adv_Arr[8] := FALSE;
   S703_TL_DC_U262_1_UP_DN.Visu_Adv_Arr[9] := FALSE;
   S703_TL_DC_U262_1_UP_DN.Visu_Adv_Arr[10] := FALSE;
   S703_TL_DC_U262_1_UP_DN.Visu_Adv_Arr[11] := FALSE;
   S703_TL_DC_U262_1_UP_DN.Visu_Adv_Arr[12] := FALSE;
   S703_TL_DC_U262_1_UP_DN.Visu_Adv_Arr[13] := FALSE;
   S703_TL_DC_U262_1_UP_DN.Visu_Adv_Arr[14] := FALSE;
   S703_TL_DC_U262_1_UP_DN.Visu_Adv_Arr[15] := FALSE;
   S703_TL_DC_U262_1_UP_DN.Visu_Ret_Arr[0] := FALSE;
   S703_TL_DC_U262_1_UP_DN.Visu_Ret_Arr[1] := FALSE;
   S703_TL_DC_U262_1_UP_DN.Visu_Ret_Arr[2] := FALSE;
   S703_TL_DC_U262_1_UP_DN.Visu_Ret_Arr[3] := FALSE;
   S703_TL_DC_U262_1_UP_DN.Visu_Ret_Arr[4] := FALSE;
   S703_TL_DC_U262_1_UP_DN.Visu_Ret_Arr[5] := FALSE;
   S703_TL_DC_U262_1_UP_DN.Visu_Ret_Arr[6] := FALSE;
   S703_TL_DC_U262_1_UP_DN.Visu_Ret_Arr[7] := FALSE;
   S703_TL_DC_U262_1_UP_DN.Visu_Ret_Arr[8] := FALSE;
   S703_TL_DC_U262_1_UP_DN.Visu_Ret_Arr[9] := FALSE;
   S703_TL_DC_U262_1_UP_DN.Visu_Ret_Arr[10] := FALSE;
   S703_TL_DC_U262_1_UP_DN.Visu_Ret_Arr[11] := FALSE;
   S703_TL_DC_U262_1_UP_DN.Visu_Ret_Arr[12] := FALSE;
   S703_TL_DC_U262_1_UP_DN.Visu_Ret_Arr[13] := FALSE;
   S703_TL_DC_U262_1_UP_DN.Visu_Ret_Arr[14] := FALSE;
   S703_TL_DC_U262_1_UP_DN.Visu_Ret_Arr[15] := FALSE;
   S703_TL_DC_U262_1_UP_DN.BLK_Move_Ret := 0;
   S703_TL_DC_U262_1_UP_DN.Enable := FALSE;
   S703_TL_DC_U262_1_UP_DN.Adv_End := FALSE;
   S703_TL_DC_U262_1_UP_DN.Ret_End := FALSE;
   S703_TL_DC_U262_1.Enable_Aux := FALSE;
   S703_TL_DC_U262_1.Adv_Amount := 0;
   S703_TL_DC_U262_1.Ret_Amount := 0;
   S703_TL_DC_U262_1.LS_Adv1 := FALSE;
   S703_TL_DC_U262_1.LS_Ret1 := FALSE;
   S703_TL_DC_U262_1.LS_Adv2 := FALSE;
   S703_TL_DC_U262_1.LS_Ret2 := FALSE;
   S703_TL_DC_U262_1.LS_Adv3 := FALSE;
   S703_TL_DC_U262_1.LS_Ret3 := FALSE;
   S703_TL_DC_U262_1.LS_Adv4 := FALSE;
   S703_TL_DC_U262_1.LS_Ret4 := FALSE;
   S703_TL_DC_U262_1.LS_Adv5 := FALSE;
   S703_TL_DC_U262_1.LS_Ret5 := FALSE;
   S703_TL_DC_U262_1.LS_Adv6 := FALSE;
   S703_TL_DC_U262_1.LS_Ret6 := FALSE;
   S703_TL_DC_U262_1.LS_Adv7 := FALSE;
   S703_TL_DC_U262_1.LS_Ret7 := FALSE;
   S703_TL_DC_U262_1.LS_Adv8 := FALSE;
   S703_TL_DC_U262_1.LS_Ret8 := FALSE;
   S703_TL_DC_U262_1.SOL_Adv := FALSE;
   S703_TL_DC_U262_1.SOL_Ret := FALSE;
   S703_TL_DC_U262_1.M_Ready := FALSE;
   S703_TL_DC_U262_1.T_CHK1 := T#0MS;
   S703_TL_DC_U262_1.T_CHK2 := T#0MS;
   S703_TL_DC_U262_1.PB_Lamp_CHK := FALSE;
   S703_TL_DC_U262_1.PB_Error_Rst := FALSE;
   S703_TL_DC_U262_1.M_FLICK := FALSE;
   S703_TL_DC_U262_1.M_Adv_Err := FALSE;
   S703_TL_DC_U262_1.M_Ret_Err := FALSE;
   S703_TL_DC_U262_1.LP_Adv := FALSE;
   S703_TL_DC_U262_1.LP_Ret := FALSE;
   S703_TL_DC_U262_1.Visu_Adv := W#16#0;
   S703_TL_DC_U262_1.Visu_Ret := W#16#0;
   S703_TL_DC_U262_1.Error_T1.IN := FALSE;
   S703_TL_DC_U262_1.Error_T1.PT := T#0MS;
   S703_TL_DC_U262_1.Error_T1.Q := FALSE;
   S703_TL_DC_U262_1.Error_T1.ET := T#0MS;
   S703_TL_DC_U262_1.Error_T1.STATE := B#16#0;
   S703_TL_DC_U262_1.Error_T1.STIME := T#0MS;
   S703_TL_DC_U262_1.Error_T1.ATIME := T#0MS;
   S703_TL_DC_U262_1.Error_T2.IN := FALSE;
   S703_TL_DC_U262_1.Error_T2.PT := T#0MS;
   S703_TL_DC_U262_1.Error_T2.Q := FALSE;
   S703_TL_DC_U262_1.Error_T2.ET := T#0MS;
   S703_TL_DC_U262_1.Error_T2.STATE := B#16#0;
   S703_TL_DC_U262_1.Error_T2.STIME := T#0MS;
   S703_TL_DC_U262_1.Error_T2.ATIME := T#0MS;
   S703_TL_DC_U262_1.Adv_End_Aux := FALSE;
   S703_TL_DC_U262_1.Ret_End_Aux := FALSE;
   S703_TL_DC_U262_1.CHK_Aux1 := FALSE;
   S703_TL_DC_U262_1.CHK_Aux2 := FALSE;
   S703_TL_DC_U262_1.Error_T1_DN := FALSE;
   S703_TL_DC_U262_1.Error_T2_DN := FALSE;
   S703_TL_DC_U262_1.Adv_Memo := FALSE;
   S703_TL_DC_U262_1.Visu_Adv_Arr[0] := FALSE;
   S703_TL_DC_U262_1.Visu_Adv_Arr[1] := FALSE;
   S703_TL_DC_U262_1.Visu_Adv_Arr[2] := FALSE;
   S703_TL_DC_U262_1.Visu_Adv_Arr[3] := FALSE;
   S703_TL_DC_U262_1.Visu_Adv_Arr[4] := FALSE;
   S703_TL_DC_U262_1.Visu_Adv_Arr[5] := FALSE;
   S703_TL_DC_U262_1.Visu_Adv_Arr[6] := FALSE;
   S703_TL_DC_U262_1.Visu_Adv_Arr[7] := FALSE;
   S703_TL_DC_U262_1.Visu_Adv_Arr[8] := FALSE;
   S703_TL_DC_U262_1.Visu_Adv_Arr[9] := FALSE;
   S703_TL_DC_U262_1.Visu_Adv_Arr[10] := FALSE;
   S703_TL_DC_U262_1.Visu_Adv_Arr[11] := FALSE;
   S703_TL_DC_U262_1.Visu_Adv_Arr[12] := FALSE;
   S703_TL_DC_U262_1.Visu_Adv_Arr[13] := FALSE;
   S703_TL_DC_U262_1.Visu_Adv_Arr[14] := FALSE;
   S703_TL_DC_U262_1.Visu_Adv_Arr[15] := FALSE;
   S703_TL_DC_U262_1.Visu_Ret_Arr[0] := FALSE;
   S703_TL_DC_U262_1.Visu_Ret_Arr[1] := FALSE;
   S703_TL_DC_U262_1.Visu_Ret_Arr[2] := FALSE;
   S703_TL_DC_U262_1.Visu_Ret_Arr[3] := FALSE;
   S703_TL_DC_U262_1.Visu_Ret_Arr[4] := FALSE;
   S703_TL_DC_U262_1.Visu_Ret_Arr[5] := FALSE;
   S703_TL_DC_U262_1.Visu_Ret_Arr[6] := FALSE;
   S703_TL_DC_U262_1.Visu_Ret_Arr[7] := FALSE;
   S703_TL_DC_U262_1.Visu_Ret_Arr[8] := FALSE;
   S703_TL_DC_U262_1.Visu_Ret_Arr[9] := FALSE;
   S703_TL_DC_U262_1.Visu_Ret_Arr[10] := FALSE;
   S703_TL_DC_U262_1.Visu_Ret_Arr[11] := FALSE;
   S703_TL_DC_U262_1.Visu_Ret_Arr[12] := FALSE;
   S703_TL_DC_U262_1.Visu_Ret_Arr[13] := FALSE;
   S703_TL_DC_U262_1.Visu_Ret_Arr[14] := FALSE;
   S703_TL_DC_U262_1.Visu_Ret_Arr[15] := FALSE;
   S703_TL_DC_U262_1.BLK_Move_Ret := 0;
   S703_TL_DC_U262_1.Enable := FALSE;
   S703_TL_DC_U262_1.Adv_End := FALSE;
   S703_TL_DC_U262_1.Ret_End := FALSE;
   S703_TL_DC_U262_1_CLAMP.Enable_Aux := FALSE;
   S703_TL_DC_U262_1_CLAMP.Adv_Amount := 0;
   S703_TL_DC_U262_1_CLAMP.Ret_Amount := 0;
   S703_TL_DC_U262_1_CLAMP.LS_Adv1 := FALSE;
   S703_TL_DC_U262_1_CLAMP.LS_Ret1 := FALSE;
   S703_TL_DC_U262_1_CLAMP.LS_Adv2 := FALSE;
   S703_TL_DC_U262_1_CLAMP.LS_Ret2 := FALSE;
   S703_TL_DC_U262_1_CLAMP.LS_Adv3 := FALSE;
   S703_TL_DC_U262_1_CLAMP.LS_Ret3 := FALSE;
   S703_TL_DC_U262_1_CLAMP.LS_Adv4 := FALSE;
   S703_TL_DC_U262_1_CLAMP.LS_Ret4 := FALSE;
   S703_TL_DC_U262_1_CLAMP.LS_Adv5 := FALSE;
   S703_TL_DC_U262_1_CLAMP.LS_Ret5 := FALSE;
   S703_TL_DC_U262_1_CLAMP.LS_Adv6 := FALSE;
   S703_TL_DC_U262_1_CLAMP.LS_Ret6 := FALSE;
   S703_TL_DC_U262_1_CLAMP.LS_Adv7 := FALSE;
   S703_TL_DC_U262_1_CLAMP.LS_Ret7 := FALSE;
   S703_TL_DC_U262_1_CLAMP.LS_Adv8 := FALSE;
   S703_TL_DC_U262_1_CLAMP.LS_Ret8 := FALSE;
   S703_TL_DC_U262_1_CLAMP.SOL_Adv := FALSE;
   S703_TL_DC_U262_1_CLAMP.SOL_Ret := FALSE;
   S703_TL_DC_U262_1_CLAMP.M_Ready := FALSE;
   S703_TL_DC_U262_1_CLAMP.T_CHK1 := T#0MS;
   S703_TL_DC_U262_1_CLAMP.T_CHK2 := T#0MS;
   S703_TL_DC_U262_1_CLAMP.PB_Lamp_CHK := FALSE;
   S703_TL_DC_U262_1_CLAMP.PB_Error_Rst := FALSE;
   S703_TL_DC_U262_1_CLAMP.M_FLICK := FALSE;
   S703_TL_DC_U262_1_CLAMP.M_Adv_Err := FALSE;
   S703_TL_DC_U262_1_CLAMP.M_Ret_Err := FALSE;
   S703_TL_DC_U262_1_CLAMP.LP_Adv := FALSE;
   S703_TL_DC_U262_1_CLAMP.LP_Ret := FALSE;
   S703_TL_DC_U262_1_CLAMP.Visu_Adv := W#16#0;
   S703_TL_DC_U262_1_CLAMP.Visu_Ret := W#16#0;
   S703_TL_DC_U262_1_CLAMP.Error_T1.IN := FALSE;
   S703_TL_DC_U262_1_CLAMP.Error_T1.PT := T#0MS;
   S703_TL_DC_U262_1_CLAMP.Error_T1.Q := FALSE;
   S703_TL_DC_U262_1_CLAMP.Error_T1.ET := T#0MS;
   S703_TL_DC_U262_1_CLAMP.Error_T1.STATE := B#16#0;
   S703_TL_DC_U262_1_CLAMP.Error_T1.STIME := T#0MS;
   S703_TL_DC_U262_1_CLAMP.Error_T1.ATIME := T#0MS;
   S703_TL_DC_U262_1_CLAMP.Error_T2.IN := FALSE;
   S703_TL_DC_U262_1_CLAMP.Error_T2.PT := T#0MS;
   S703_TL_DC_U262_1_CLAMP.Error_T2.Q := FALSE;
   S703_TL_DC_U262_1_CLAMP.Error_T2.ET := T#0MS;
   S703_TL_DC_U262_1_CLAMP.Error_T2.STATE := B#16#0;
   S703_TL_DC_U262_1_CLAMP.Error_T2.STIME := T#0MS;
   S703_TL_DC_U262_1_CLAMP.Error_T2.ATIME := T#0MS;
   S703_TL_DC_U262_1_CLAMP.Adv_End_Aux := FALSE;
   S703_TL_DC_U262_1_CLAMP.Ret_End_Aux := FALSE;
   S703_TL_DC_U262_1_CLAMP.CHK_Aux1 := FALSE;
   S703_TL_DC_U262_1_CLAMP.CHK_Aux2 := FALSE;
   S703_TL_DC_U262_1_CLAMP.Error_T1_DN := FALSE;
   S703_TL_DC_U262_1_CLAMP.Error_T2_DN := FALSE;
   S703_TL_DC_U262_1_CLAMP.Adv_Memo := FALSE;
   S703_TL_DC_U262_1_CLAMP.Visu_Adv_Arr[0] := FALSE;
   S703_TL_DC_U262_1_CLAMP.Visu_Adv_Arr[1] := FALSE;
   S703_TL_DC_U262_1_CLAMP.Visu_Adv_Arr[2] := FALSE;
   S703_TL_DC_U262_1_CLAMP.Visu_Adv_Arr[3] := FALSE;
   S703_TL_DC_U262_1_CLAMP.Visu_Adv_Arr[4] := FALSE;
   S703_TL_DC_U262_1_CLAMP.Visu_Adv_Arr[5] := FALSE;
   S703_TL_DC_U262_1_CLAMP.Visu_Adv_Arr[6] := FALSE;
   S703_TL_DC_U262_1_CLAMP.Visu_Adv_Arr[7] := FALSE;
   S703_TL_DC_U262_1_CLAMP.Visu_Adv_Arr[8] := FALSE;
   S703_TL_DC_U262_1_CLAMP.Visu_Adv_Arr[9] := FALSE;
   S703_TL_DC_U262_1_CLAMP.Visu_Adv_Arr[10] := FALSE;
   S703_TL_DC_U262_1_CLAMP.Visu_Adv_Arr[11] := FALSE;
   S703_TL_DC_U262_1_CLAMP.Visu_Adv_Arr[12] := FALSE;
   S703_TL_DC_U262_1_CLAMP.Visu_Adv_Arr[13] := FALSE;
   S703_TL_DC_U262_1_CLAMP.Visu_Adv_Arr[14] := FALSE;
   S703_TL_DC_U262_1_CLAMP.Visu_Adv_Arr[15] := FALSE;
   S703_TL_DC_U262_1_CLAMP.Visu_Ret_Arr[0] := FALSE;
   S703_TL_DC_U262_1_CLAMP.Visu_Ret_Arr[1] := FALSE;
   S703_TL_DC_U262_1_CLAMP.Visu_Ret_Arr[2] := FALSE;
   S703_TL_DC_U262_1_CLAMP.Visu_Ret_Arr[3] := FALSE;
   S703_TL_DC_U262_1_CLAMP.Visu_Ret_Arr[4] := FALSE;
   S703_TL_DC_U262_1_CLAMP.Visu_Ret_Arr[5] := FALSE;
   S703_TL_DC_U262_1_CLAMP.Visu_Ret_Arr[6] := FALSE;
   S703_TL_DC_U262_1_CLAMP.Visu_Ret_Arr[7] := FALSE;
   S703_TL_DC_U262_1_CLAMP.Visu_Ret_Arr[8] := FALSE;
   S703_TL_DC_U262_1_CLAMP.Visu_Ret_Arr[9] := FALSE;
   S703_TL_DC_U262_1_CLAMP.Visu_Ret_Arr[10] := FALSE;
   S703_TL_DC_U262_1_CLAMP.Visu_Ret_Arr[11] := FALSE;
   S703_TL_DC_U262_1_CLAMP.Visu_Ret_Arr[12] := FALSE;
   S703_TL_DC_U262_1_CLAMP.Visu_Ret_Arr[13] := FALSE;
   S703_TL_DC_U262_1_CLAMP.Visu_Ret_Arr[14] := FALSE;
   S703_TL_DC_U262_1_CLAMP.Visu_Ret_Arr[15] := FALSE;
   S703_TL_DC_U262_1_CLAMP.BLK_Move_Ret := 0;
   S703_TL_DC_U262_1_CLAMP.Enable := FALSE;
   S703_TL_DC_U262_1_CLAMP.Adv_End := FALSE;
   S703_TL_DC_U262_1_CLAMP.Ret_End := FALSE;
   S703_TL_DC_U261_2_CLAMP.Enable_Aux := FALSE;
   S703_TL_DC_U261_2_CLAMP.Adv_Amount := 0;
   S703_TL_DC_U261_2_CLAMP.Ret_Amount := 0;
   S703_TL_DC_U261_2_CLAMP.LS_Adv1 := FALSE;
   S703_TL_DC_U261_2_CLAMP.LS_Ret1 := FALSE;
   S703_TL_DC_U261_2_CLAMP.LS_Adv2 := FALSE;
   S703_TL_DC_U261_2_CLAMP.LS_Ret2 := FALSE;
   S703_TL_DC_U261_2_CLAMP.LS_Adv3 := FALSE;
   S703_TL_DC_U261_2_CLAMP.LS_Ret3 := FALSE;
   S703_TL_DC_U261_2_CLAMP.LS_Adv4 := FALSE;
   S703_TL_DC_U261_2_CLAMP.LS_Ret4 := FALSE;
   S703_TL_DC_U261_2_CLAMP.LS_Adv5 := FALSE;
   S703_TL_DC_U261_2_CLAMP.LS_Ret5 := FALSE;
   S703_TL_DC_U261_2_CLAMP.LS_Adv6 := FALSE;
   S703_TL_DC_U261_2_CLAMP.LS_Ret6 := FALSE;
   S703_TL_DC_U261_2_CLAMP.LS_Adv7 := FALSE;
   S703_TL_DC_U261_2_CLAMP.LS_Ret7 := FALSE;
   S703_TL_DC_U261_2_CLAMP.LS_Adv8 := FALSE;
   S703_TL_DC_U261_2_CLAMP.LS_Ret8 := FALSE;
   S703_TL_DC_U261_2_CLAMP.SOL_Adv := FALSE;
   S703_TL_DC_U261_2_CLAMP.SOL_Ret := FALSE;
   S703_TL_DC_U261_2_CLAMP.M_Ready := FALSE;
   S703_TL_DC_U261_2_CLAMP.T_CHK1 := T#0MS;
   S703_TL_DC_U261_2_CLAMP.T_CHK2 := T#0MS;
   S703_TL_DC_U261_2_CLAMP.PB_Lamp_CHK := FALSE;
   S703_TL_DC_U261_2_CLAMP.PB_Error_Rst := FALSE;
   S703_TL_DC_U261_2_CLAMP.M_FLICK := FALSE;
   S703_TL_DC_U261_2_CLAMP.M_Adv_Err := FALSE;
   S703_TL_DC_U261_2_CLAMP.M_Ret_Err := FALSE;
   S703_TL_DC_U261_2_CLAMP.LP_Adv := FALSE;
   S703_TL_DC_U261_2_CLAMP.LP_Ret := FALSE;
   S703_TL_DC_U261_2_CLAMP.Visu_Adv := W#16#0;
   S703_TL_DC_U261_2_CLAMP.Visu_Ret := W#16#0;
   S703_TL_DC_U261_2_CLAMP.Error_T1.IN := FALSE;
   S703_TL_DC_U261_2_CLAMP.Error_T1.PT := T#0MS;
   S703_TL_DC_U261_2_CLAMP.Error_T1.Q := FALSE;
   S703_TL_DC_U261_2_CLAMP.Error_T1.ET := T#0MS;
   S703_TL_DC_U261_2_CLAMP.Error_T1.STATE := B#16#0;
   S703_TL_DC_U261_2_CLAMP.Error_T1.STIME := T#0MS;
   S703_TL_DC_U261_2_CLAMP.Error_T1.ATIME := T#0MS;
   S703_TL_DC_U261_2_CLAMP.Error_T2.IN := FALSE;
   S703_TL_DC_U261_2_CLAMP.Error_T2.PT := T#0MS;
   S703_TL_DC_U261_2_CLAMP.Error_T2.Q := FALSE;
   S703_TL_DC_U261_2_CLAMP.Error_T2.ET := T#0MS;
   S703_TL_DC_U261_2_CLAMP.Error_T2.STATE := B#16#0;
   S703_TL_DC_U261_2_CLAMP.Error_T2.STIME := T#0MS;
   S703_TL_DC_U261_2_CLAMP.Error_T2.ATIME := T#0MS;
   S703_TL_DC_U261_2_CLAMP.Adv_End_Aux := FALSE;
   S703_TL_DC_U261_2_CLAMP.Ret_End_Aux := FALSE;
   S703_TL_DC_U261_2_CLAMP.CHK_Aux1 := FALSE;
   S703_TL_DC_U261_2_CLAMP.CHK_Aux2 := FALSE;
   S703_TL_DC_U261_2_CLAMP.Error_T1_DN := FALSE;
   S703_TL_DC_U261_2_CLAMP.Error_T2_DN := FALSE;
   S703_TL_DC_U261_2_CLAMP.Adv_Memo := FALSE;
   S703_TL_DC_U261_2_CLAMP.Visu_Adv_Arr[0] := FALSE;
   S703_TL_DC_U261_2_CLAMP.Visu_Adv_Arr[1] := FALSE;
   S703_TL_DC_U261_2_CLAMP.Visu_Adv_Arr[2] := FALSE;
   S703_TL_DC_U261_2_CLAMP.Visu_Adv_Arr[3] := FALSE;
   S703_TL_DC_U261_2_CLAMP.Visu_Adv_Arr[4] := FALSE;
   S703_TL_DC_U261_2_CLAMP.Visu_Adv_Arr[5] := FALSE;
   S703_TL_DC_U261_2_CLAMP.Visu_Adv_Arr[6] := FALSE;
   S703_TL_DC_U261_2_CLAMP.Visu_Adv_Arr[7] := FALSE;
   S703_TL_DC_U261_2_CLAMP.Visu_Adv_Arr[8] := FALSE;
   S703_TL_DC_U261_2_CLAMP.Visu_Adv_Arr[9] := FALSE;
   S703_TL_DC_U261_2_CLAMP.Visu_Adv_Arr[10] := FALSE;
   S703_TL_DC_U261_2_CLAMP.Visu_Adv_Arr[11] := FALSE;
   S703_TL_DC_U261_2_CLAMP.Visu_Adv_Arr[12] := FALSE;
   S703_TL_DC_U261_2_CLAMP.Visu_Adv_Arr[13] := FALSE;
   S703_TL_DC_U261_2_CLAMP.Visu_Adv_Arr[14] := FALSE;
   S703_TL_DC_U261_2_CLAMP.Visu_Adv_Arr[15] := FALSE;
   S703_TL_DC_U261_2_CLAMP.Visu_Ret_Arr[0] := FALSE;
   S703_TL_DC_U261_2_CLAMP.Visu_Ret_Arr[1] := FALSE;
   S703_TL_DC_U261_2_CLAMP.Visu_Ret_Arr[2] := FALSE;
   S703_TL_DC_U261_2_CLAMP.Visu_Ret_Arr[3] := FALSE;
   S703_TL_DC_U261_2_CLAMP.Visu_Ret_Arr[4] := FALSE;
   S703_TL_DC_U261_2_CLAMP.Visu_Ret_Arr[5] := FALSE;
   S703_TL_DC_U261_2_CLAMP.Visu_Ret_Arr[6] := FALSE;
   S703_TL_DC_U261_2_CLAMP.Visu_Ret_Arr[7] := FALSE;
   S703_TL_DC_U261_2_CLAMP.Visu_Ret_Arr[8] := FALSE;
   S703_TL_DC_U261_2_CLAMP.Visu_Ret_Arr[9] := FALSE;
   S703_TL_DC_U261_2_CLAMP.Visu_Ret_Arr[10] := FALSE;
   S703_TL_DC_U261_2_CLAMP.Visu_Ret_Arr[11] := FALSE;
   S703_TL_DC_U261_2_CLAMP.Visu_Ret_Arr[12] := FALSE;
   S703_TL_DC_U261_2_CLAMP.Visu_Ret_Arr[13] := FALSE;
   S703_TL_DC_U261_2_CLAMP.Visu_Ret_Arr[14] := FALSE;
   S703_TL_DC_U261_2_CLAMP.Visu_Ret_Arr[15] := FALSE;
   S703_TL_DC_U261_2_CLAMP.BLK_Move_Ret := 0;
   S703_TL_DC_U261_2_CLAMP.Enable := FALSE;
   S703_TL_DC_U261_2_CLAMP.Adv_End := FALSE;
   S703_TL_DC_U261_2_CLAMP.Ret_End := FALSE;
END_DATA_BLOCK

FUNCTION FC 134 : VOID
TITLE =
VERSION : 0.1

BEGIN
NETWORK
TITLE =
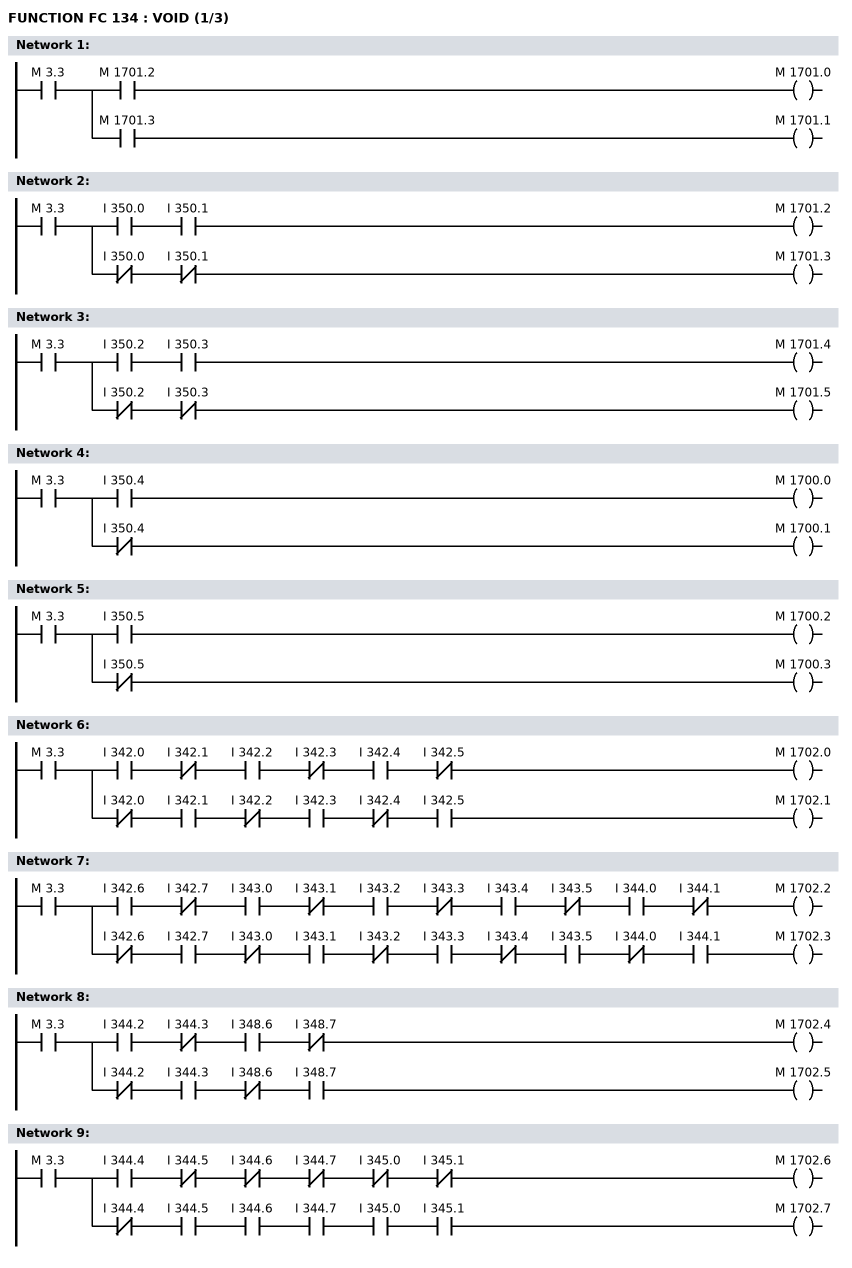

      A     M      3.3;
      =     L      0.0;
      A     L      0.0;
      A     M   1701.2;
      =     M   1701.0;
      A     L      0.0;
      A     M   1701.3;
      =     M   1701.1;
NETWORK
TITLE =

      A     M      3.3;
      =     L      0.0;
      A     L      0.0;
      A     I    350.0;
      A     I    350.1;
      =     M   1701.2;
      A     L      0.0;
      AN    I    350.0;
      AN    I    350.1;
      =     M   1701.3;
NETWORK
TITLE =

      A     M      3.3;
      =     L      0.0;
      A     L      0.0;
      A     I    350.2;
      A     I    350.3;
      =     M   1701.4;
      A     L      0.0;
      AN    I    350.2;
      AN    I    350.3;
      =     M   1701.5;
NETWORK
TITLE =

      A     M      3.3;
      =     L      0.0;
      A     L      0.0;
      A     I    350.4;
      =     M   1700.0;
      A     L      0.0;
      AN    I    350.4;
      =     M   1700.1;
NETWORK
TITLE =

      A     M      3.3;
      =     L      0.0;
      A     L      0.0;
      A     I    350.5;
      =     M   1700.2;
      A     L      0.0;
      AN    I    350.5;
      =     M   1700.3;
NETWORK
TITLE =

      A     M      3.3;
      =     L      0.0;
      A     L      0.0;
      A     I    342.0;
      AN    I    342.1;
      A     I    342.2;
      AN    I    342.3;
      A     I    342.4;
      AN    I    342.5;
      =     M   1702.0;
      A     L      0.0;
      AN    I    342.0;
      A     I    342.1;
      AN    I    342.2;
      A     I    342.3;
      AN    I    342.4;
      A     I    342.5;
      =     M   1702.1;
NETWORK
TITLE =

      A     M      3.3;
      =     L      0.0;
      A     L      0.0;
      A     I    342.6;
      AN    I    342.7;
      A     I    343.0;
      AN    I    343.1;
      A     I    343.2;
      AN    I    343.3;
      A     I    343.4;
      AN    I    343.5;
      A     I    344.0;
      AN    I    344.1;
      =     M   1702.2;
      A     L      0.0;
      AN    I    342.6;
      A     I    342.7;
      AN    I    343.0;
      A     I    343.1;
      AN    I    343.2;
      A     I    343.3;
      AN    I    343.4;
      A     I    343.5;
      AN    I    344.0;
      A     I    344.1;
      =     M   1702.3;
NETWORK
TITLE =

      A     M      3.3;
      =     L      0.0;
      A     L      0.0;
      A     I    344.2;
      AN    I    344.3;
      A     I    348.6;
      AN    I    348.7;
      =     M   1702.4;
      A     L      0.0;
      AN    I    344.2;
      A     I    344.3;
      AN    I    348.6;
      A     I    348.7;
      =     M   1702.5;
NETWORK
TITLE =

      A     M      3.3;
      =     L      0.0;
      A     L      0.0;
      A     I    344.4;
      AN    I    344.5;
      AN    I    344.6;
      AN    I    344.7;
      AN    I    345.0;
      AN    I    345.1;
      =     M   1702.6;
      A     L      0.0;
      AN    I    344.4;
      A     I    344.5;
      A     I    344.6;
      A     I    344.7;
      A     I    345.0;
      A     I    345.1;
      =     M   1702.7;
NETWORK
TITLE =
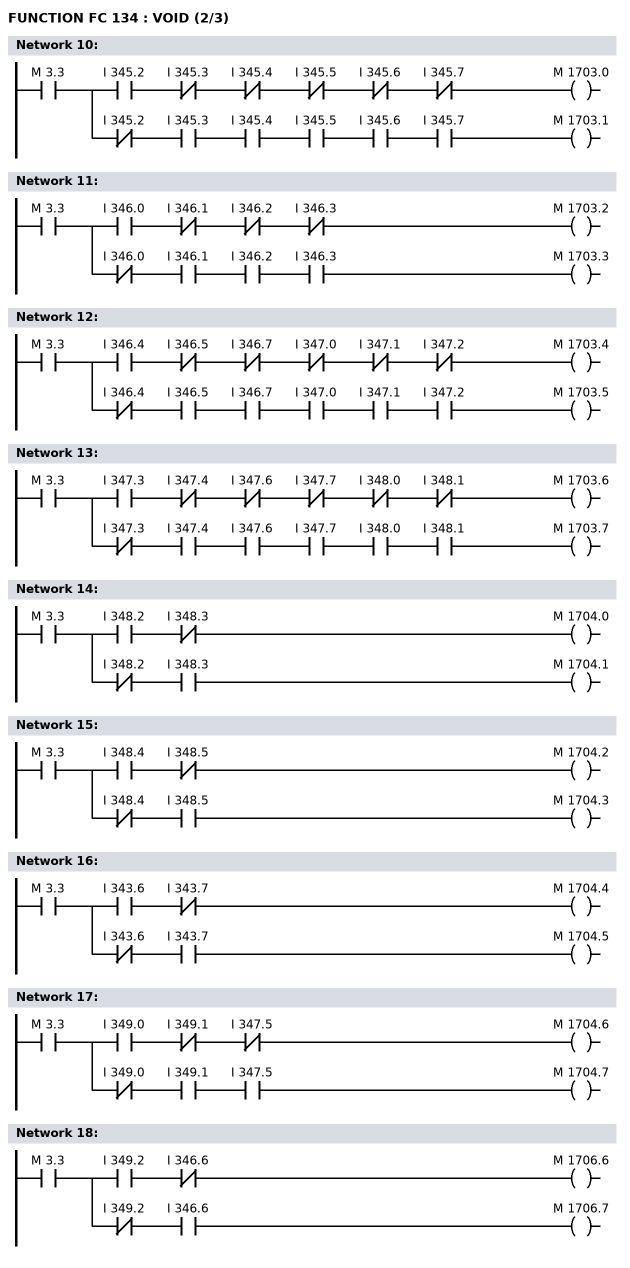

      A     M      3.3;
      =     L      0.0;
      A     L      0.0;
      A     I    345.2;
      AN    I    345.3;
      AN    I    345.4;
      AN    I    345.5;
      AN    I    345.6;
      AN    I    345.7;
      =     M   1703.0;
      A     L      0.0;
      AN    I    345.2;
      A     I    345.3;
      A     I    345.4;
      A     I    345.5;
      A     I    345.6;
      A     I    345.7;
      =     M   1703.1;
NETWORK
TITLE =

      A     M      3.3;
      =     L      0.0;
      A     L      0.0;
      A     I    346.0;
      AN    I    346.1;
      AN    I    346.2;
      AN    I    346.3;
      =     M   1703.2;
      A     L      0.0;
      AN    I    346.0;
      A     I    346.1;
      A     I    346.2;
      A     I    346.3;
      =     M   1703.3;
NETWORK
TITLE =

      A     M      3.3;
      =     L      0.0;
      A     L      0.0;
      A     I    346.4;
      AN    I    346.5;
      AN    I    346.7;
      AN    I    347.0;
      AN    I    347.1;
      AN    I    347.2;
      =     M   1703.4;
      A     L      0.0;
      AN    I    346.4;
      A     I    346.5;
      A     I    346.7;
      A     I    347.0;
      A     I    347.1;
      A     I    347.2;
      =     M   1703.5;
NETWORK
TITLE =

      A     M      3.3;
      =     L      0.0;
      A     L      0.0;
      A     I    347.3;
      AN    I    347.4;
      AN    I    347.6;
      AN    I    347.7;
      AN    I    348.0;
      AN    I    348.1;
      =     M   1703.6;
      A     L      0.0;
      AN    I    347.3;
      A     I    347.4;
      A     I    347.6;
      A     I    347.7;
      A     I    348.0;
      A     I    348.1;
      =     M   1703.7;
NETWORK
TITLE =

      A     M      3.3;
      =     L      0.0;
      A     L      0.0;
      A     I    348.2;
      AN    I    348.3;
      =     M   1704.0;
      A     L      0.0;
      AN    I    348.2;
      A     I    348.3;
      =     M   1704.1;
NETWORK
TITLE =

      A     M      3.3;
      =     L      0.0;
      A     L      0.0;
      A     I    348.4;
      AN    I    348.5;
      =     M   1704.2;
      A     L      0.0;
      AN    I    348.4;
      A     I    348.5;
      =     M   1704.3;
NETWORK
TITLE =

      A     M      3.3;
      =     L      0.0;
      A     L      0.0;
      A     I    343.6;
      AN    I    343.7;
      =     M   1704.4;
      A     L      0.0;
      AN    I    343.6;
      A     I    343.7;
      =     M   1704.5;
NETWORK
TITLE =

      A     M      3.3;
      =     L      0.0;
      A     L      0.0;
      A     I    349.0;
      AN    I    349.1;
      AN    I    347.5;
      =     M   1704.6;
      A     L      0.0;
      AN    I    349.0;
      A     I    349.1;
      A     I    347.5;
      =     M   1704.7;
NETWORK
TITLE =

      A     M      3.3;
      =     L      0.0;
      A     L      0.0;
      A     I    349.2;
      AN    I    346.6;
      =     M   1706.6;
      A     L      0.0;
      AN    I    349.2;
      A     I    346.6;
      =     M   1706.7;
NETWORK
TITLE =
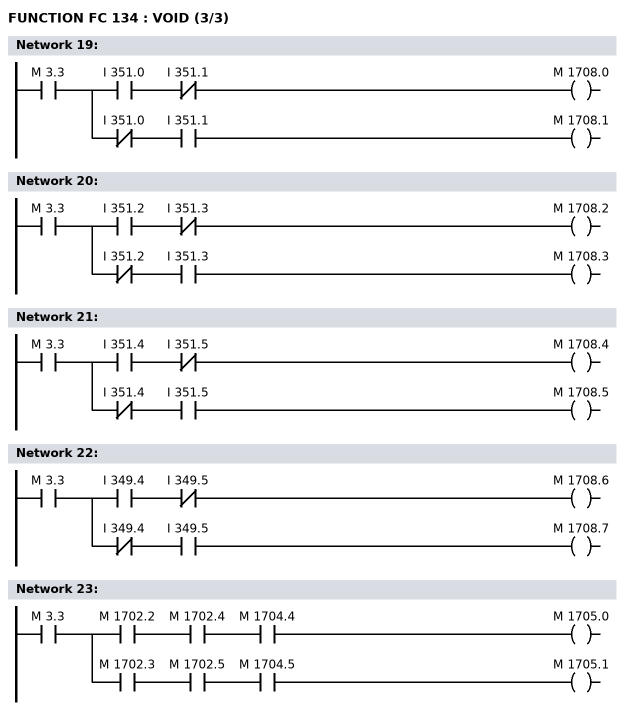

      A     M      3.3;
      =     L      0.0;
      A     L      0.0;
      A     I    351.0;
      AN    I    351.1;
      =     M   1708.0;
      A     L      0.0;
      AN    I    351.0;
      A     I    351.1;
      =     M   1708.1;
NETWORK
TITLE =

      A     M      3.3;
      =     L      0.0;
      A     L      0.0;
      A     I    351.2;
      AN    I    351.3;
      =     M   1708.2;
      A     L      0.0;
      AN    I    351.2;
      A     I    351.3;
      =     M   1708.3;
NETWORK
TITLE =

      A     M      3.3;
      =     L      0.0;
      A     L      0.0;
      A     I    351.4;
      AN    I    351.5;
      =     M   1708.4;
      A     L      0.0;
      AN    I    351.4;
      A     I    351.5;
      =     M   1708.5;
NETWORK
TITLE =

      A     M      3.3;
      =     L      0.0;
      A     L      0.0;
      A     I    349.4;
      AN    I    349.5;
      =     M   1708.6;
      A     L      0.0;
      AN    I    349.4;
      A     I    349.5;
      =     M   1708.7;
NETWORK
TITLE =

      A     M      3.3;
      =     L      0.0;
      A     L      0.0;
      A     M   1702.2;
      A     M   1702.4;
      A     M   1704.4;
      =     M   1705.0;
      A     L      0.0;
      A     M   1702.3;
      A     M   1702.5;
      A     M   1704.5;
      =     M   1705.1;
NETWORK
TITLE =

      A     M      3.3;
      =     L      0.0;
      A     L      0.0;
      A     M   1702.6;
      A     M   1703.0;
      A     M   1703.2;
      A     M   1703.4;
      A     M   1703.6;
      A     M   1706.6;
      =     L      0.1;
      A     L      0.1;
      BLD   102;
      =     M   1705.2;
      A     L      0.1;
      A     M   1704.2;
      A     M   1704.6;
      =     M   1705.4;
      A     L      0.0;
      A     M   1702.7;
      A     M   1703.1;
      A     M   1703.3;
      A     M   1703.5;
      A     M   1703.7;
      A     M   1706.7;
      =     L      0.1;
      A     L      0.1;
      BLD   102;
      =     M   1705.3;
      A     L      0.1;
      A     M   1704.3;
      A     M   1704.7;
      =     M   1705.5;
NETWORK
TITLE =
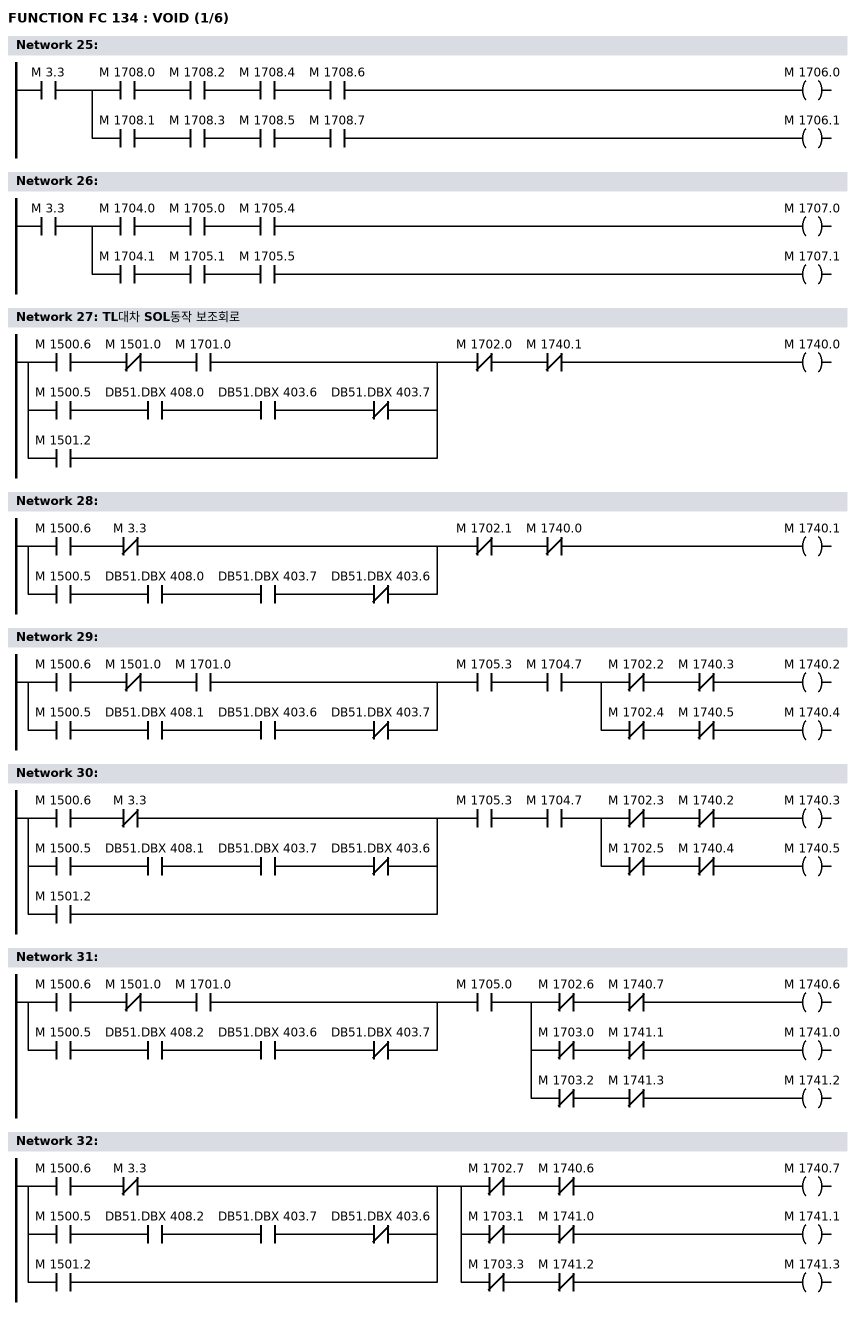

      A     M      3.3;
      =     L      0.0;
      A     L      0.0;
      A     M   1708.0;
      A     M   1708.2;
      A     M   1708.4;
      A     M   1708.6;
      =     M   1706.0;
      A     L      0.0;
      A     M   1708.1;
      A     M   1708.3;
      A     M   1708.5;
      A     M   1708.7;
      =     M   1706.1;
NETWORK
TITLE =

      A     M      3.3;
      =     L      0.0;
      A     L      0.0;
      A     M   1704.0;
      A     M   1705.0;
      A     M   1705.4;
      =     M   1707.0;
      A     L      0.0;
      A     M   1704.1;
      A     M   1705.1;
      A     M   1705.5;
      =     M   1707.1;
NETWORK
TITLE =TL대차 SOL동작 보조회로

      A(    ;
      A     M   1500.6;
      AN    M   1501.0;
      A     M   1701.0;
      O     ;
      A     M   1500.5;
      A     DB51.DBX  408.0;
      A     DB51.DBX  403.6;
      AN    DB51.DBX  403.7;
      O     M   1501.2;
      )     ;
      AN    M   1702.0;
      AN    M   1740.1;
      =     M   1740.0;
NETWORK
TITLE =

      A(    ;
      A     M   1500.6;
      AN    M      3.3;
      O     ;
      A     M   1500.5;
      A     DB51.DBX  408.0;
      A     DB51.DBX  403.7;
      AN    DB51.DBX  403.6;
      )     ;
      AN    M   1702.1;
      AN    M   1740.0;
      =     M   1740.1;
NETWORK
TITLE =

      A(    ;
      A     M   1500.6;
      AN    M   1501.0;
      A     M   1701.0;
      O     ;
      A     M   1500.5;
      A     DB51.DBX  408.1;
      A     DB51.DBX  403.6;
      AN    DB51.DBX  403.7;
      )     ;
      A     M   1705.3;
      A     M   1704.7;
      =     L      0.0;
      A     L      0.0;
      AN    M   1702.2;
      AN    M   1740.3;
      =     M   1740.2;
      A     L      0.0;
      AN    M   1702.4;
      AN    M   1740.5;
      =     M   1740.4;
NETWORK
TITLE =

      A(    ;
      A     M   1500.6;
      AN    M      3.3;
      O     ;
      A     M   1500.5;
      A     DB51.DBX  408.1;
      A     DB51.DBX  403.7;
      AN    DB51.DBX  403.6;
      O     M   1501.2;
      )     ;
      A     M   1705.3;
      A     M   1704.7;
      =     L      0.0;
      A     L      0.0;
      AN    M   1702.3;
      AN    M   1740.2;
      =     M   1740.3;
      A     L      0.0;
      AN    M   1702.5;
      AN    M   1740.4;
      =     M   1740.5;
NETWORK
TITLE =

      A(    ;
      A     M   1500.6;
      AN    M   1501.0;
      A     M   1701.0;
      O     ;
      A     M   1500.5;
      A     DB51.DBX  408.2;
      A     DB51.DBX  403.6;
      AN    DB51.DBX  403.7;
      )     ;
      A     M   1705.0;
      =     L      0.0;
      A     L      0.0;
      AN    M   1702.6;
      AN    M   1740.7;
      =     M   1740.6;
      A     L      0.0;
      AN    M   1703.0;
      AN    M   1741.1;
      =     M   1741.0;
      A     L      0.0;
      AN    M   1703.2;
      AN    M   1741.3;
      =     M   1741.2;
NETWORK
TITLE =

      A     M   1500.6;
      AN    M      3.3;
      O     ;
      A     M   1500.5;
      A     DB51.DBX  408.2;
      A     DB51.DBX  403.7;
      AN    DB51.DBX  403.6;
      O     M   1501.2;
      =     L      0.0;
      A     L      0.0;
      AN    M   1702.7;
      AN    M   1740.6;
      =     M   1740.7;
      A     L      0.0;
      AN    M   1703.1;
      AN    M   1741.0;
      =     M   1741.1;
      A     L      0.0;
      AN    M   1703.3;
      AN    M   1741.2;
      =     M   1741.3;
NETWORK
TITLE =
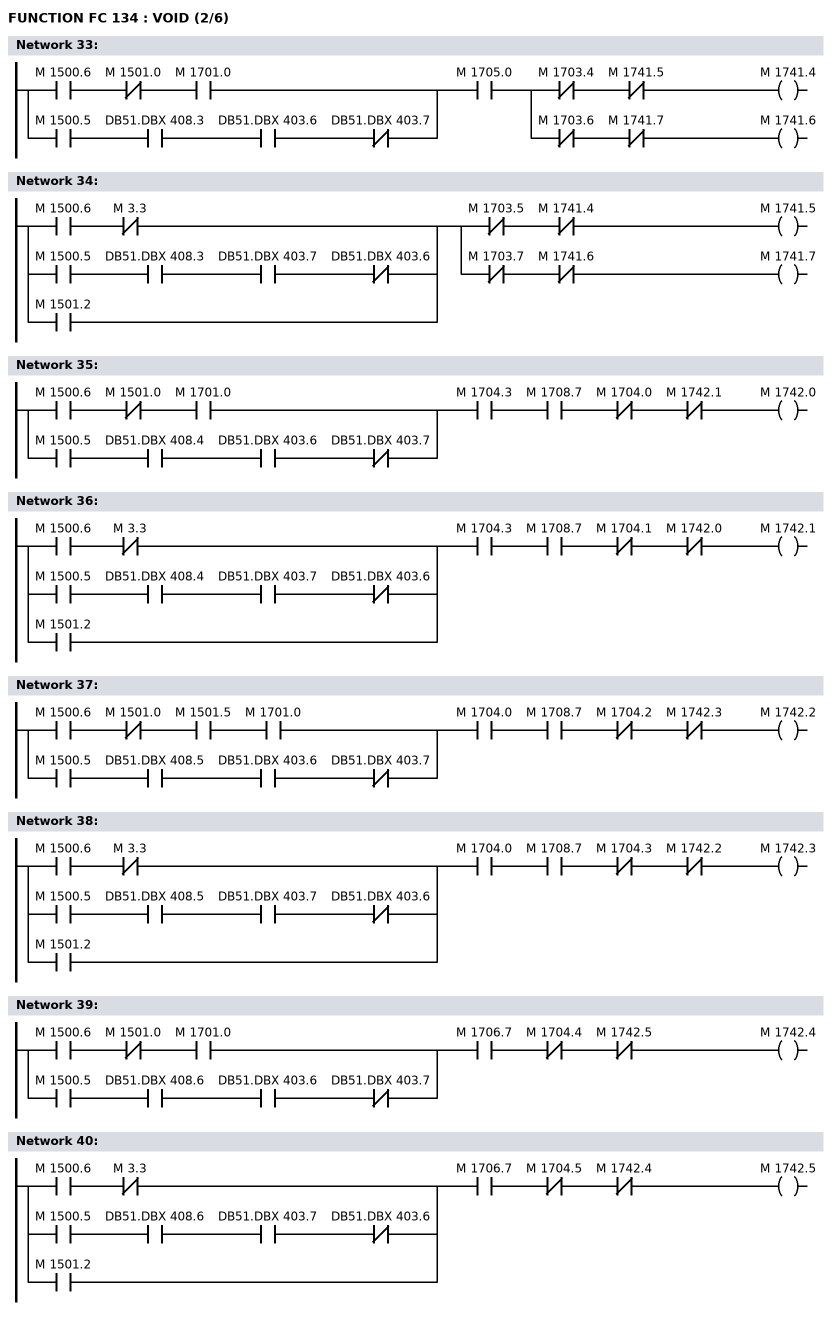

      A(    ;
      A     M   1500.6;
      AN    M   1501.0;
      A     M   1701.0;
      O     ;
      A     M   1500.5;
      A     DB51.DBX  408.3;
      A     DB51.DBX  403.6;
      AN    DB51.DBX  403.7;
      )     ;
      A     M   1705.0;
      =     L      0.0;
      A     L      0.0;
      AN    M   1703.4;
      AN    M   1741.5;
      =     M   1741.4;
      A     L      0.0;
      AN    M   1703.6;
      AN    M   1741.7;
      =     M   1741.6;
NETWORK
TITLE =

      A     M   1500.6;
      AN    M      3.3;
      O     ;
      A     M   1500.5;
      A     DB51.DBX  408.3;
      A     DB51.DBX  403.7;
      AN    DB51.DBX  403.6;
      O     M   1501.2;
      =     L      0.0;
      A     L      0.0;
      AN    M   1703.5;
      AN    M   1741.4;
      =     M   1741.5;
      A     L      0.0;
      AN    M   1703.7;
      AN    M   1741.6;
      =     M   1741.7;
NETWORK
TITLE =

      A(    ;
      A     M   1500.6;
      AN    M   1501.0;
      A     M   1701.0;
      O     ;
      A     M   1500.5;
      A     DB51.DBX  408.4;
      A     DB51.DBX  403.6;
      AN    DB51.DBX  403.7;
      )     ;
      A     M   1704.3;
      A     M   1708.7;
      AN    M   1704.0;
      AN    M   1742.1;
      =     M   1742.0;
NETWORK
TITLE =

      A(    ;
      A     M   1500.6;
      AN    M      3.3;
      O     ;
      A     M   1500.5;
      A     DB51.DBX  408.4;
      A     DB51.DBX  403.7;
      AN    DB51.DBX  403.6;
      O     M   1501.2;
      )     ;
      A     M   1704.3;
      A     M   1708.7;
      AN    M   1704.1;
      AN    M   1742.0;
      =     M   1742.1;
NETWORK
TITLE =

      A(    ;
      A     M   1500.6;
      AN    M   1501.0;
      A     M   1501.5;
      A     M   1701.0;
      O     ;
      A     M   1500.5;
      A     DB51.DBX  408.5;
      A     DB51.DBX  403.6;
      AN    DB51.DBX  403.7;
      )     ;
      A     M   1704.0;
      A     M   1708.7;
      AN    M   1704.2;
      AN    M   1742.3;
      =     M   1742.2;
NETWORK
TITLE =

      A(    ;
      A     M   1500.6;
      AN    M      3.3;
      O     ;
      A     M   1500.5;
      A     DB51.DBX  408.5;
      A     DB51.DBX  403.7;
      AN    DB51.DBX  403.6;
      O     M   1501.2;
      )     ;
      A     M   1704.0;
      A     M   1708.7;
      AN    M   1704.3;
      AN    M   1742.2;
      =     M   1742.3;
NETWORK
TITLE =

      A(    ;
      A     M   1500.6;
      AN    M   1501.0;
      A     M   1701.0;
      O     ;
      A     M   1500.5;
      A     DB51.DBX  408.6;
      A     DB51.DBX  403.6;
      AN    DB51.DBX  403.7;
      )     ;
      A     M   1706.7;
      AN    M   1704.4;
      AN    M   1742.5;
      =     M   1742.4;
NETWORK
TITLE =

      A(    ;
      A     M   1500.6;
      AN    M      3.3;
      O     ;
      A     M   1500.5;
      A     DB51.DBX  408.6;
      A     DB51.DBX  403.7;
      AN    DB51.DBX  403.6;
      O     M   1501.2;
      )     ;
      A     M   1706.7;
      AN    M   1704.5;
      AN    M   1742.4;
      =     M   1742.5;
NETWORK
TITLE =
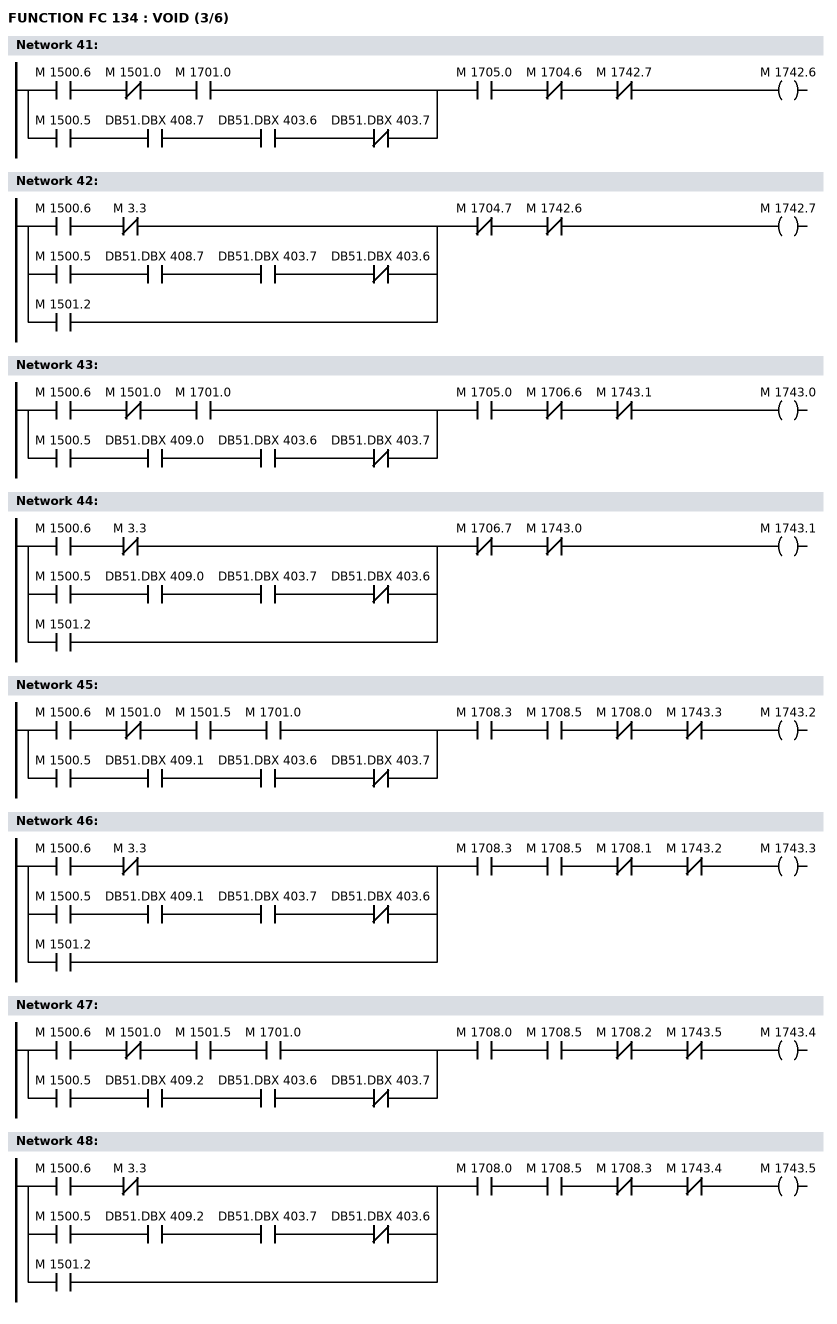

      A(    ;
      A     M   1500.6;
      AN    M   1501.0;
      A     M   1701.0;
      O     ;
      A     M   1500.5;
      A     DB51.DBX  408.7;
      A     DB51.DBX  403.6;
      AN    DB51.DBX  403.7;
      )     ;
      A     M   1705.0;
      AN    M   1704.6;
      AN    M   1742.7;
      =     M   1742.6;
NETWORK
TITLE =

      A(    ;
      A     M   1500.6;
      AN    M      3.3;
      O     ;
      A     M   1500.5;
      A     DB51.DBX  408.7;
      A     DB51.DBX  403.7;
      AN    DB51.DBX  403.6;
      O     M   1501.2;
      )     ;
      AN    M   1704.7;
      AN    M   1742.6;
      =     M   1742.7;
NETWORK
TITLE =

      A(    ;
      A     M   1500.6;
      AN    M   1501.0;
      A     M   1701.0;
      O     ;
      A     M   1500.5;
      A     DB51.DBX  409.0;
      A     DB51.DBX  403.6;
      AN    DB51.DBX  403.7;
      )     ;
      A     M   1705.0;
      AN    M   1706.6;
      AN    M   1743.1;
      =     M   1743.0;
NETWORK
TITLE =

      A(    ;
      A     M   1500.6;
      AN    M      3.3;
      O     ;
      A     M   1500.5;
      A     DB51.DBX  409.0;
      A     DB51.DBX  403.7;
      AN    DB51.DBX  403.6;
      O     M   1501.2;
      )     ;
      AN    M   1706.7;
      AN    M   1743.0;
      =     M   1743.1;
NETWORK
TITLE =

      A(    ;
      A     M   1500.6;
      AN    M   1501.0;
      A     M   1501.5;
      A     M   1701.0;
      O     ;
      A     M   1500.5;
      A     DB51.DBX  409.1;
      A     DB51.DBX  403.6;
      AN    DB51.DBX  403.7;
      )     ;
      A     M   1708.3;
      A     M   1708.5;
      AN    M   1708.0;
      AN    M   1743.3;
      =     M   1743.2;
NETWORK
TITLE =

      A(    ;
      A     M   1500.6;
      AN    M      3.3;
      O     ;
      A     M   1500.5;
      A     DB51.DBX  409.1;
      A     DB51.DBX  403.7;
      AN    DB51.DBX  403.6;
      O     M   1501.2;
      )     ;
      A     M   1708.3;
      A     M   1708.5;
      AN    M   1708.1;
      AN    M   1743.2;
      =     M   1743.3;
NETWORK
TITLE =

      A(    ;
      A     M   1500.6;
      AN    M   1501.0;
      A     M   1501.5;
      A     M   1701.0;
      O     ;
      A     M   1500.5;
      A     DB51.DBX  409.2;
      A     DB51.DBX  403.6;
      AN    DB51.DBX  403.7;
      )     ;
      A     M   1708.0;
      A     M   1708.5;
      AN    M   1708.2;
      AN    M   1743.5;
      =     M   1743.4;
NETWORK
TITLE =

      A(    ;
      A     M   1500.6;
      AN    M      3.3;
      O     ;
      A     M   1500.5;
      A     DB51.DBX  409.2;
      A     DB51.DBX  403.7;
      AN    DB51.DBX  403.6;
      O     M   1501.2;
      )     ;
      A     M   1708.0;
      A     M   1708.5;
      AN    M   1708.3;
      AN    M   1743.4;
      =     M   1743.5;
NETWORK
TITLE =
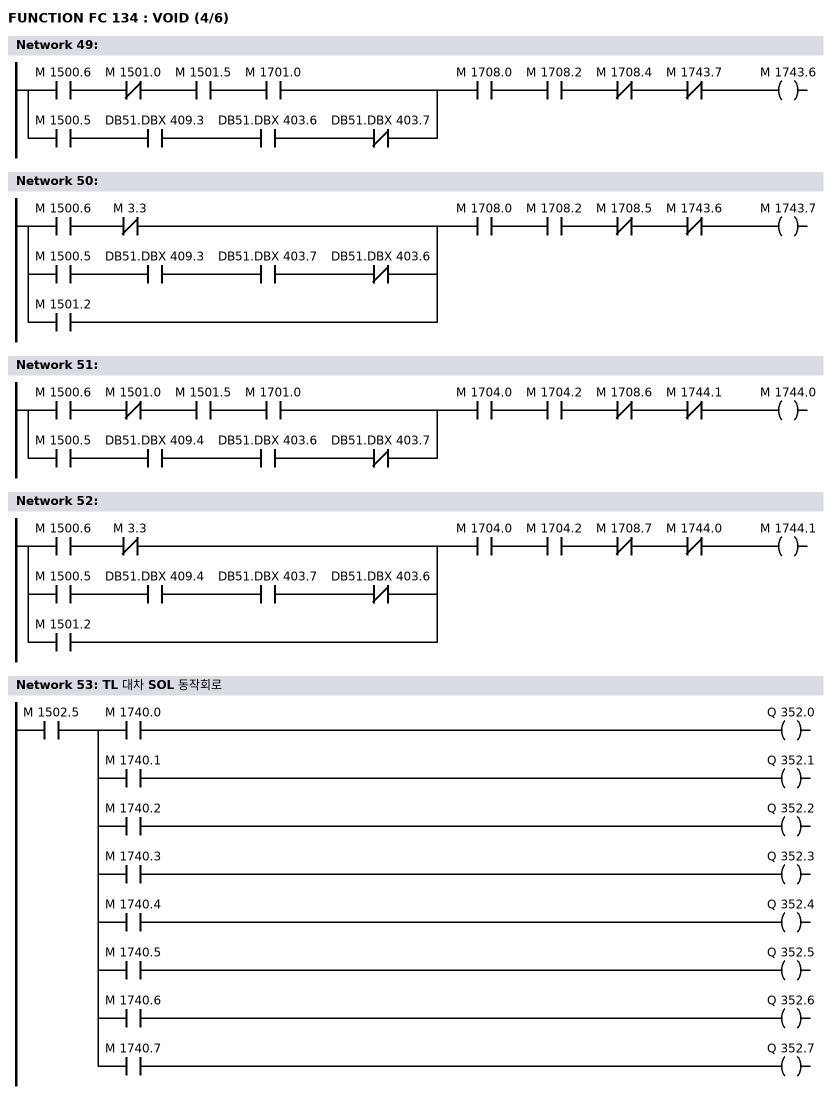

      A(    ;
      A     M   1500.6;
      AN    M   1501.0;
      A     M   1501.5;
      A     M   1701.0;
      O     ;
      A     M   1500.5;
      A     DB51.DBX  409.3;
      A     DB51.DBX  403.6;
      AN    DB51.DBX  403.7;
      )     ;
      A     M   1708.0;
      A     M   1708.2;
      AN    M   1708.4;
      AN    M   1743.7;
      =     M   1743.6;
NETWORK
TITLE =

      A(    ;
      A     M   1500.6;
      AN    M      3.3;
      O     ;
      A     M   1500.5;
      A     DB51.DBX  409.3;
      A     DB51.DBX  403.7;
      AN    DB51.DBX  403.6;
      O     M   1501.2;
      )     ;
      A     M   1708.0;
      A     M   1708.2;
      AN    M   1708.5;
      AN    M   1743.6;
      =     M   1743.7;
NETWORK
TITLE =

      A(    ;
      A     M   1500.6;
      AN    M   1501.0;
      A     M   1501.5;
      A     M   1701.0;
      O     ;
      A     M   1500.5;
      A     DB51.DBX  409.4;
      A     DB51.DBX  403.6;
      AN    DB51.DBX  403.7;
      )     ;
      A     M   1704.0;
      A     M   1704.2;
      AN    M   1708.6;
      AN    M   1744.1;
      =     M   1744.0;
NETWORK
TITLE =

      A(    ;
      A     M   1500.6;
      AN    M      3.3;
      O     ;
      A     M   1500.5;
      A     DB51.DBX  409.4;
      A     DB51.DBX  403.7;
      AN    DB51.DBX  403.6;
      O     M   1501.2;
      )     ;
      A     M   1704.0;
      A     M   1704.2;
      AN    M   1708.7;
      AN    M   1744.0;
      =     M   1744.1;
NETWORK
TITLE =TL 대차 SOL 동작회로

      A     M   1502.5;
      =     L      0.0;
      A     L      0.0;
      A     M   1740.0;
      =     Q    352.0;
      A     L      0.0;
      A     M   1740.1;
      =     Q    352.1;
      A     L      0.0;
      A     M   1740.2;
      =     Q    352.2;
      A     L      0.0;
      A     M   1740.3;
      =     Q    352.3;
      A     L      0.0;
      A     M   1740.4;
      =     Q    352.4;
      A     L      0.0;
      A     M   1740.5;
      =     Q    352.5;
      A     L      0.0;
      A     M   1740.6;
      =     Q    352.6;
      A     L      0.0;
      A     M   1740.7;
      =     Q    352.7;
NETWORK
TITLE =
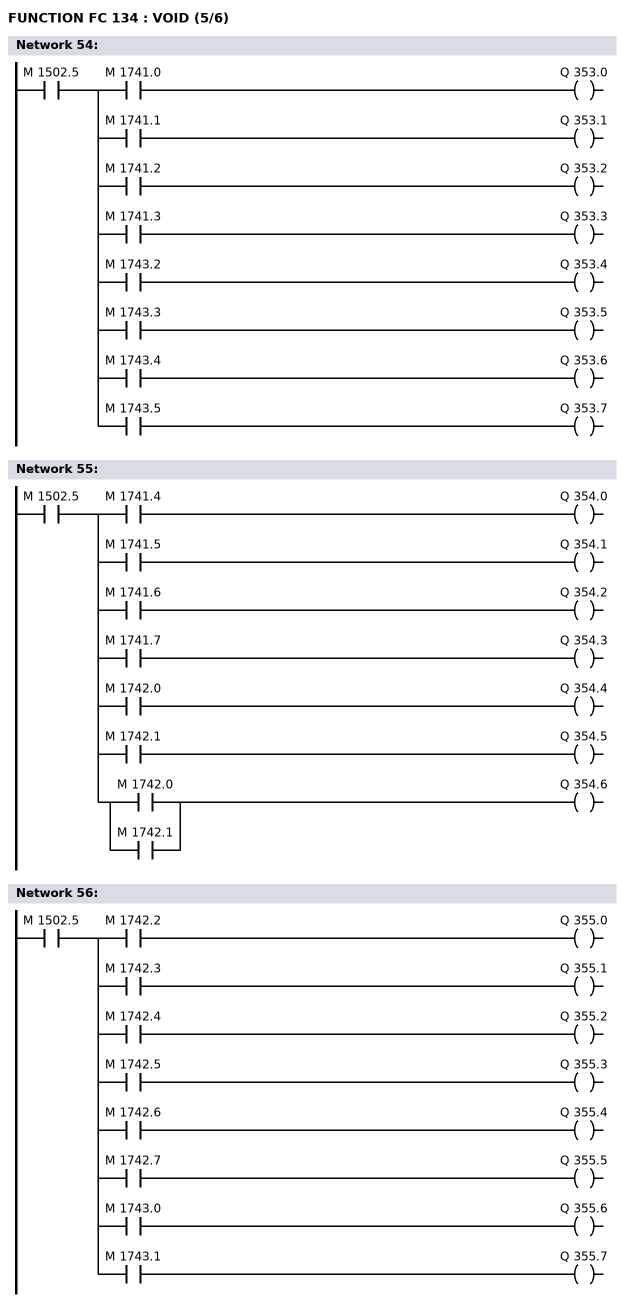

      A     M   1502.5;
      =     L      0.0;
      A     L      0.0;
      A     M   1741.0;
      =     Q    353.0;
      A     L      0.0;
      A     M   1741.1;
      =     Q    353.1;
      A     L      0.0;
      A     M   1741.2;
      =     Q    353.2;
      A     L      0.0;
      A     M   1741.3;
      =     Q    353.3;
      A     L      0.0;
      A     M   1743.2;
      =     Q    353.4;
      A     L      0.0;
      A     M   1743.3;
      =     Q    353.5;
      A     L      0.0;
      A     M   1743.4;
      =     Q    353.6;
      A     L      0.0;
      A     M   1743.5;
      =     Q    353.7;
NETWORK
TITLE =

      A     M   1502.5;
      =     L      0.0;
      A     L      0.0;
      A     M   1741.4;
      =     Q    354.0;
      A     L      0.0;
      A     M   1741.5;
      =     Q    354.1;
      A     L      0.0;
      A     M   1741.6;
      =     Q    354.2;
      A     L      0.0;
      A     M   1741.7;
      =     Q    354.3;
      A     L      0.0;
      A     M   1742.0;
      =     Q    354.4;
      A     L      0.0;
      A     M   1742.1;
      =     Q    354.5;
      A     L      0.0;
      A(    ;
      O     M   1742.0;
      O     M   1742.1;
      )     ;
      =     Q    354.6;
NETWORK
TITLE =

      A     M   1502.5;
      =     L      0.0;
      A     L      0.0;
      A     M   1742.2;
      =     Q    355.0;
      A     L      0.0;
      A     M   1742.3;
      =     Q    355.1;
      A     L      0.0;
      A     M   1742.4;
      =     Q    355.2;
      A     L      0.0;
      A     M   1742.5;
      =     Q    355.3;
      A     L      0.0;
      A     M   1742.6;
      =     Q    355.4;
      A     L      0.0;
      A     M   1742.7;
      =     Q    355.5;
      A     L      0.0;
      A     M   1743.0;
      =     Q    355.6;
      A     L      0.0;
      A     M   1743.1;
      =     Q    355.7;
NETWORK
TITLE =
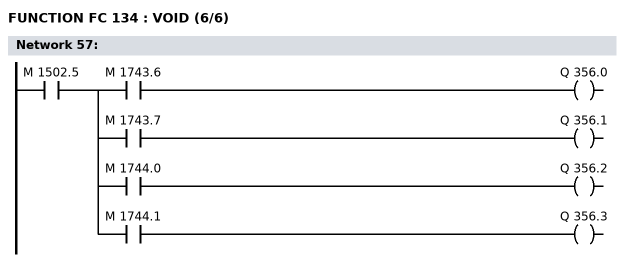

      A     M   1502.5;
      =     L      0.0;
      A     L      0.0;
      A     M   1743.6;
      =     Q    356.0;
      A     L      0.0;
      A     M   1743.7;
      =     Q    356.1;
      A     L      0.0;
      A     M   1744.0;
      =     Q    356.2;
      A     L      0.0;
      A     M   1744.1;
      =     Q    356.3;
END_FUNCTION

FUNCTION_BLOCK FB 140
TITLE =
VERSION : 0.1


VAR
  S704_MODE : FB 402;
END_VAR
BEGIN
NETWORK
TITLE =
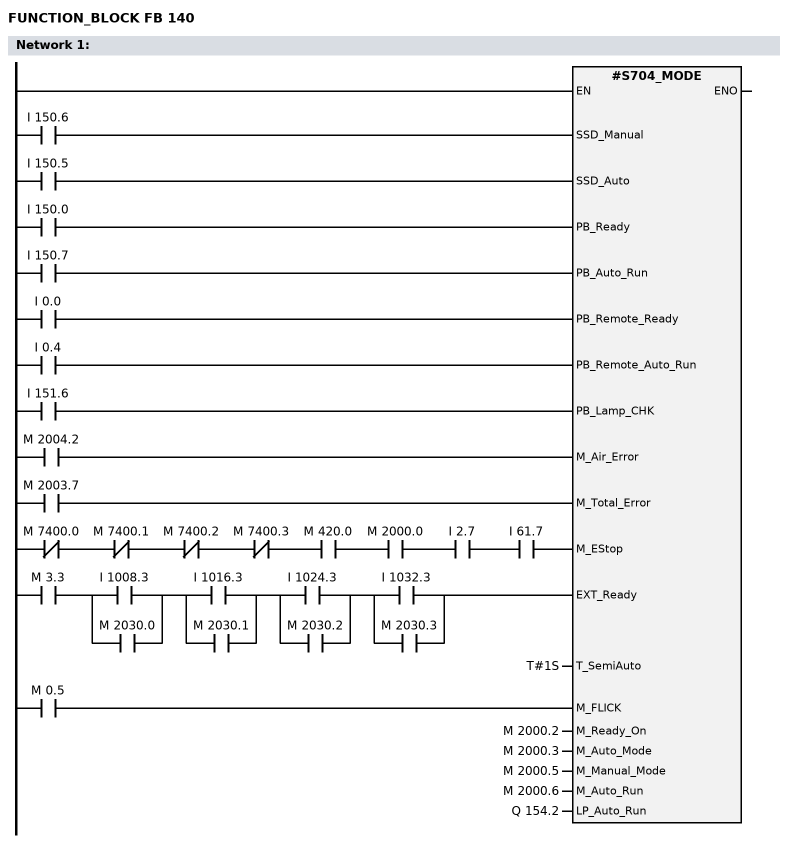

      A     I    150.6;
      =     L      0.0;
      BLD   103;
      A     I    150.5;
      =     L      0.1;
      BLD   103;
      A     I    150.0;
      =     L      0.2;
      BLD   103;
      A     I    150.7;
      =     L      0.3;
      BLD   103;
      A     I      0.0;
      =     L      0.4;
      BLD   103;
      A     I      0.4;
      =     L      0.5;
      BLD   103;
      A     I    151.6;
      =     L      0.6;
      BLD   103;
      A     M   2004.2;
      =     L      0.7;
      BLD   103;
      A     M   2003.7;
      =     L      1.1;
      BLD   103;
      AN    M   7400.0;
      AN    M   7400.1;
      AN    M   7400.2;
      AN    M   7400.3;
      A     M    420.0;
      A     M   2000.0;
      A     I      2.7;
      A     I     61.7;
      =     L      1.2;
      BLD   103;
      A     M      3.3;
      A(    ;
      O     I   1008.3;
      O     M   2030.0;
      )     ;
      A(    ;
      O     I   1016.3;
      O     M   2030.1;
      )     ;
      A(    ;
      O     I   1024.3;
      O     M   2030.2;
      )     ;
      A(    ;
      O     I   1032.3;
      O     M   2030.3;
      )     ;
      =     L      1.3;
      BLD   103;
      A     M      0.5;
      =     L      1.5;
      BLD   103;
      CALL #S704_MODE (
           SSD_Manual               := L      0.0,
           SSD_Auto                 := L      0.1,
           PB_Ready                 := L      0.2,
           PB_Auto_Run              := L      0.3,
           PB_Remote_Ready          := L      0.4,
           PB_Remote_Auto_Run       := L      0.5,
           PB_Lamp_CHK              := L      0.6,
           M_Air_Error              := L      0.7,
           M_Total_Error            := L      1.1,
           M_EStop                  := L      1.2,
           EXT_Ready                := L      1.3,
           T_SemiAuto               := T#1S,
           M_FLICK                  := L      1.5,
           M_Ready_On               := M   2000.2,
           M_Auto_Mode              := M   2000.3,
           M_Manual_Mode            := M   2000.5,
           M_Auto_Run               := M   2000.6,
           LP_Auto_Run              := Q    154.2);
      NOP   0;
END_FUNCTION_BLOCK

DATA_BLOCK DB 140
TITLE =
VERSION : 0.0

 FB 140
BEGIN
   S704_MODE.SSD_Manual := FALSE;
   S704_MODE.SSD_Auto := FALSE;
   S704_MODE.PB_Ready := FALSE;
   S704_MODE.PB_Auto_Run := FALSE;
   S704_MODE.PB_Remote_Ready := FALSE;
   S704_MODE.PB_Remote_Auto_Run := FALSE;
   S704_MODE.PB_Lamp_CHK := FALSE;
   S704_MODE.M_Air_Error := FALSE;
   S704_MODE.M_Water_Error := FALSE;
   S704_MODE.M_Total_Error := FALSE;
   S704_MODE.M_EStop := FALSE;
   S704_MODE.EXT_Ready := FALSE;
   S704_MODE.EXT_Auto := FALSE;
   S704_MODE.T_SemiAuto := T#0MS;
   S704_MODE.M_FLICK := FALSE;
   S704_MODE.M_Ready_On := FALSE;
   S704_MODE.M_Auto_Mode := FALSE;
   S704_MODE.M_SemiAuto_Mode := FALSE;
   S704_MODE.M_Manual_Mode := FALSE;
   S704_MODE.M_Auto_Run := FALSE;
   S704_MODE.LP_Ready_On := FALSE;
   S704_MODE.LP_Auto_Run := FALSE;
   S704_MODE.AUTO_MODE_DELAY.IN := FALSE;
   S704_MODE.AUTO_MODE_DELAY.PT := T#0MS;
   S704_MODE.AUTO_MODE_DELAY.Q := FALSE;
   S704_MODE.AUTO_MODE_DELAY.ET := T#0MS;
   S704_MODE.AUTO_MODE_DELAY.STATE := B#16#0;
   S704_MODE.AUTO_MODE_DELAY.STIME := T#0MS;
   S704_MODE.AUTO_MODE_DELAY.ATIME := T#0MS;
   S704_MODE.SEMI_AUTO_DELAY.IN := FALSE;
   S704_MODE.SEMI_AUTO_DELAY.PT := T#0MS;
   S704_MODE.SEMI_AUTO_DELAY.Q := FALSE;
   S704_MODE.SEMI_AUTO_DELAY.ET := T#0MS;
   S704_MODE.SEMI_AUTO_DELAY.STATE := B#16#0;
   S704_MODE.SEMI_AUTO_DELAY.STIME := T#0MS;
   S704_MODE.SEMI_AUTO_DELAY.ATIME := T#0MS;
   S704_MODE.MANUAL_DELAY.IN := FALSE;
   S704_MODE.MANUAL_DELAY.PT := T#0MS;
   S704_MODE.MANUAL_DELAY.Q := FALSE;
   S704_MODE.MANUAL_DELAY.ET := T#0MS;
   S704_MODE.MANUAL_DELAY.STATE := B#16#0;
   S704_MODE.MANUAL_DELAY.STIME := T#0MS;
   S704_MODE.MANUAL_DELAY.ATIME := T#0MS;
END_DATA_BLOCK

FUNCTION FC 140 : VOID
TITLE =
VERSION : 0.1

BEGIN
NETWORK
TITLE =
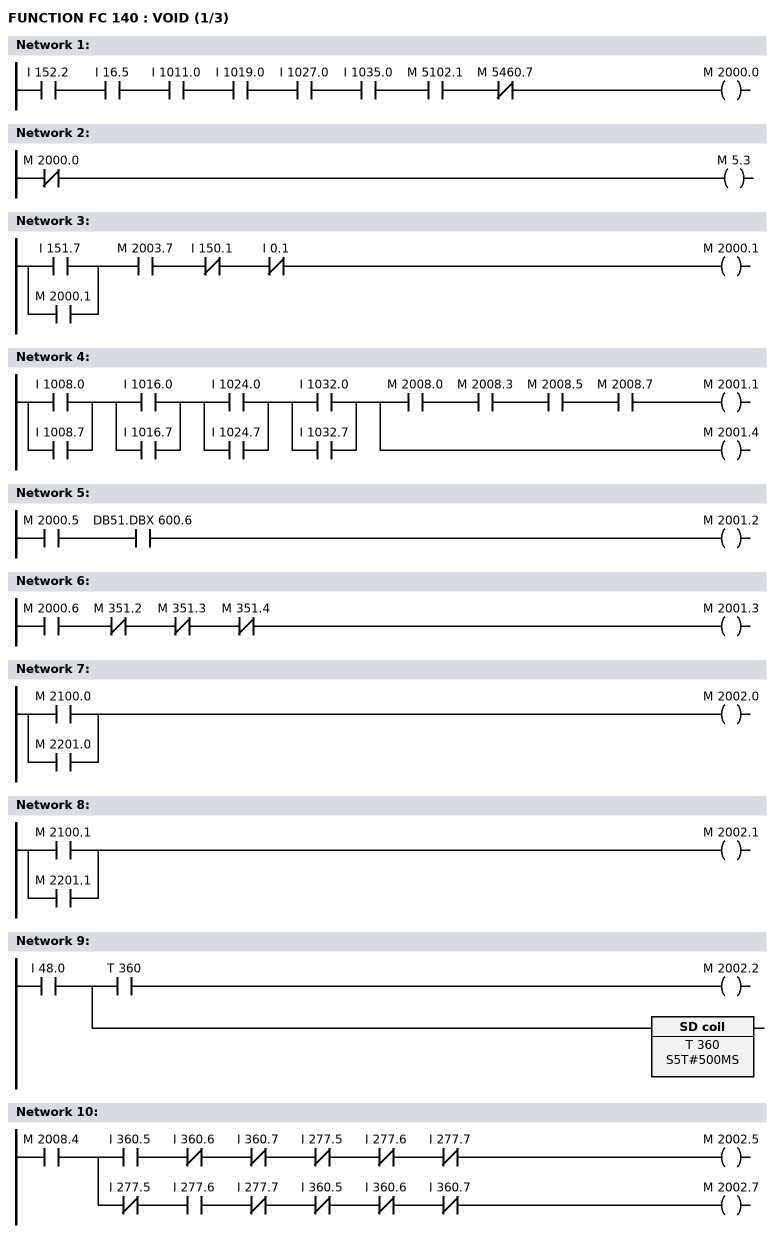

      A     I    152.2;
      A     I     16.5;
      A     I   1011.0;
      A     I   1019.0;
      A     I   1027.0;
      A     I   1035.0;
      A     M   5102.1;
      AN    M   5460.7;
      =     M   2000.0;
NETWORK
TITLE =

      AN    M   2000.0;
      =     M      5.3;
NETWORK
TITLE =

      A(    ;
      O     I    151.7;
      O     M   2000.1;
      )     ;
      A     M   2003.7;
      AN    I    150.1;
      AN    I      0.1;
      =     M   2000.1;
NETWORK
TITLE =

      A(    ;
      O     I   1008.0;
      O     I   1008.7;
      )     ;
      A(    ;
      O     I   1016.0;
      O     I   1016.7;
      )     ;
      A(    ;
      O     I   1024.0;
      O     I   1024.7;
      )     ;
      A(    ;
      O     I   1032.0;
      O     I   1032.7;
      )     ;
      =     L      0.0;
      A     L      0.0;
      A     M   2008.0;
      A     M   2008.3;
      A     M   2008.5;
      A     M   2008.7;
      =     M   2001.1;
      A     L      0.0;
      BLD   102;
      =     M   2001.4;
NETWORK
TITLE =

      A     M   2000.5;
      A     DB51.DBX  600.6;
      =     M   2001.2;
NETWORK
TITLE =

      A     M   2000.6;
      AN    M    351.2;
      AN    M    351.3;
      AN    M    351.4;
      =     M   2001.3;
NETWORK
TITLE =

      O     M   2100.0;
      O     M   2201.0;
      =     M   2002.0;
NETWORK
TITLE =

      O     M   2100.1;
      O     M   2201.1;
      =     M   2002.1;
NETWORK
TITLE =

      A     I     48.0;
      =     L      0.0;
      A     L      0.0;
      A     T    360;
      =     M   2002.2;
      A     L      0.0;
      BLD   102;
      L     S5T#500MS;
      SD    T    360;
NETWORK
TITLE =

      A     M   2008.4;
      =     L      0.0;
      A     L      0.0;
      A     I    360.5;
      AN    I    360.6;
      AN    I    360.7;
      AN    I    277.5;
      AN    I    277.6;
      AN    I    277.7;
      =     M   2002.5;
      A     L      0.0;
      AN    I    277.5;
      A     I    277.6;
      AN    I    277.7;
      AN    I    360.5;
      AN    I    360.6;
      AN    I    360.7;
      =     M   2002.7;
NETWORK
TITLE =
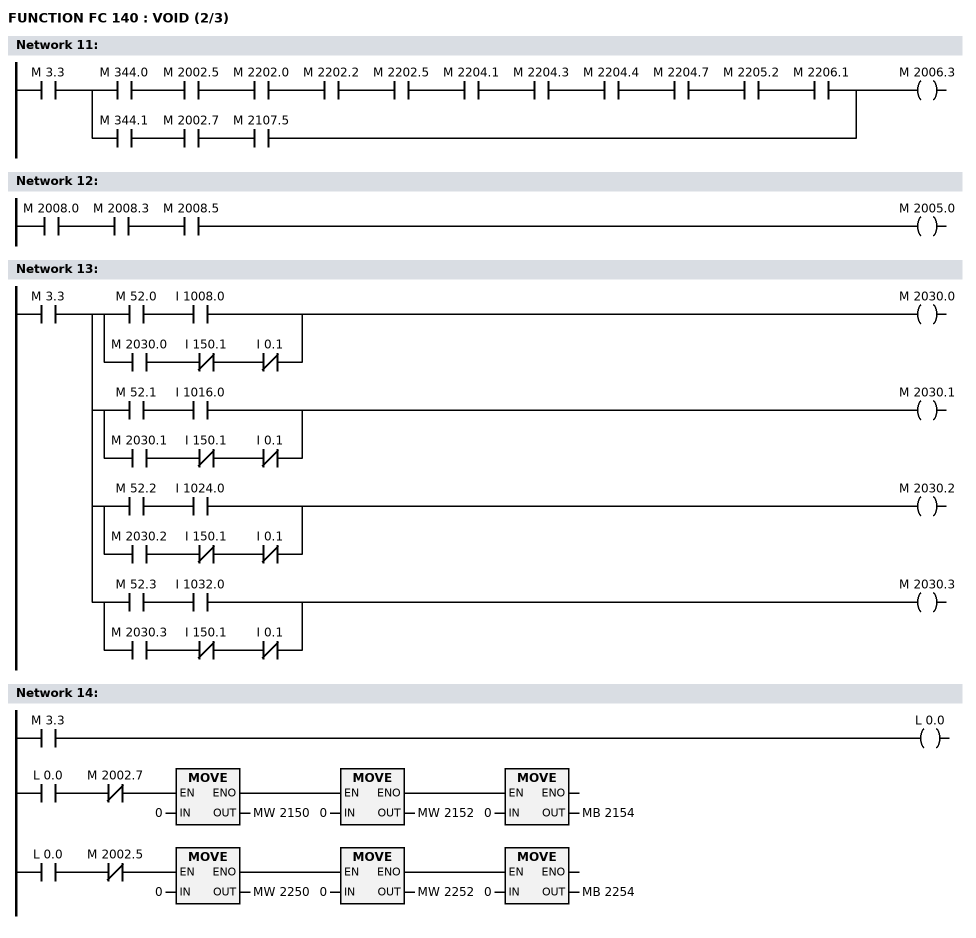

      A     M      3.3;
      A(    ;
      A     M    344.0;
      A     M   2002.5;
      A     M   2202.0;
      A     M   2202.2;
      A     M   2202.5;
      A     M   2204.1;
      A     M   2204.3;
      A     M   2204.4;
      A     M   2204.7;
      A     M   2205.2;
      A     M   2206.1;
      O     ;
      A     M    344.1;
      A     M   2002.7;
      A     M   2107.5;
      )     ;
      =     M   2006.3;
NETWORK
TITLE =

      A     M   2008.0;
      A     M   2008.3;
      A     M   2008.5;
      =     M   2005.0;
NETWORK
TITLE =

      A     M      3.3;
      =     L      0.0;
      A     L      0.0;
      A(    ;
      A     M     52.0;
      A     I   1008.0;
      O     ;
      A     M   2030.0;
      AN    I    150.1;
      AN    I      0.1;
      )     ;
      =     M   2030.0;
      A     L      0.0;
      A(    ;
      A     M     52.1;
      A     I   1016.0;
      O     ;
      A     M   2030.1;
      AN    I    150.1;
      AN    I      0.1;
      )     ;
      =     M   2030.1;
      A     L      0.0;
      A(    ;
      A     M     52.2;
      A     I   1024.0;
      O     ;
      A     M   2030.2;
      AN    I    150.1;
      AN    I      0.1;
      )     ;
      =     M   2030.2;
      A     L      0.0;
      A(    ;
      A     M     52.3;
      A     I   1032.0;
      O     ;
      A     M   2030.3;
      AN    I    150.1;
      AN    I      0.1;
      )     ;
      =     M   2030.3;
NETWORK
TITLE =

